LIN {X 0,Y 256.186,Z 305.925,A -85,B 0,C 180,E1 -18988.035,E2 -18988.035} C_VEL
LIN {X 0,Y 254.625,Z 317.423,A -85,B 0,C 180,E1 -18989.605,E2 -18989.605} C_VEL
LIN {X 0,Y 253.092,Z 328.163,A -85,B 0,C 180,E1 -18991.482,E2 -18991.482} C_VEL
LIN {X 0,Y 251.484,Z 337.845,A -85,B 0,C 180,E1 -18993.605,E2 -18993.605} C_VEL
LIN {X 0,Y 250.27,Z 345.355,A -85,B 0,C 180,E1 -18995.641,E2 -18995.641} C_VEL
LIN {X 0,Y 249.076,Z 352.738,A -85,B 0,C 180,E1 -18998.111,E2 -18998.111} C_VEL
LIN {X 0,Y 248.18,Z 358.597,A -85,B 0,C 180,E1 -19000.607,E2 -19000.607} C_VEL
LIN {X 0,Y 247.564,Z 363.197,A -85,B 0,C 180,E1 -19003.127,E2 -19003.127} C_VEL
LIN {X 0,Y 247.222,Z 365.688,A -85,B 0,C 180,E1 -19004.863,E2 -19004.863} C_VEL
LIN {X 0,Y 246.962,Z 367.629,A -85,B 0,C 180,E1 -19006.534,E2 -19006.534} C_VEL
LIN {X 0,Y 246.859,Z 369.106,A -85,B 0,C 180,E1 -19008.25,E2 -19008.25} C_VEL
LIN {X 0,Y 246.842,Z 370.181,A -85,B 0,C 180,E1 -19010.022,E2 -19010.022} C_VEL
LIN {X 0,Y 246.907,Z 370.793,A -85,B 0,C 180,E1 -19011.718,E2 -19011.718} C_VEL
LIN {X 0,Y 247.304,Z 370.822,A -85,B 0,C 180,E1 -19014.579,E2 -19014.579} C_VEL
LIN {X 0,Y 247.898,Z 369.931,A -85,B 0,C 180,E1 -19016.976,E2 -19016.976} C_VEL
LIN {X 0,Y 248.543,Z 368.668,A -85,B 0,C 180,E1 -19018.768,E2 -19018.768} C_VEL
LIN {X 0,Y 249.722,Z 365.952,A -85,B 0,C 180,E1 -19021.376,E2 -19021.376} C_VEL
LIN {X 0,Y 251.297,Z 362.009,A -85,B 0,C 180,E1 -19024.01,E2 -19024.01} C_VEL
LIN {X 0,Y 253.501,Z 356.251,A -85,B 0,C 180,E1 -19026.834,E2 -19026.834} C_VEL
LIN {X 0,Y 255.77,Z 349.911,A -85,B 0,C 180,E1 -19029.197,E2 -19029.197} C_VEL
LIN {X 0,Y 258.193,Z 342.787,A -85,B 0,C 180,E1 -19031.307,E2 -19031.307} C_VEL
LIN {X 0,Y 260.783,Z 334.381,A -85,B 0,C 180,E1 -19033.312,E2 -19033.312} C_VEL
LIN {X 0,Y 263.669,Z 324.355,A -85,B 0,C 180,E1 -19035.209,E2 -19035.209} C_VEL
LIN {X 0,Y 266.207,Z 314.054,A -85,B 0,C 180,E1 -19036.755,E2 -19036.755} C_VEL
LIN {X 0,Y 268.658,Z 301.667,A -85,B 0,C 180,E1 -19038.207,E2 -19038.207} C_VEL
LIN {X 0,Y 270.547,Z 289.737,A -85,B 0,C 180,E1 -19039.262,E2 -19039.262} C_VEL
LIN {X 0,Y 271.947,Z 277.419,A -85,B 0,C 180,E1 -19040.048,E2 -19040.048} C_VEL
LIN {X 0,Y 272.934,Z 264.372,A -85,B 0,C 180,E1 -19040.579,E2 -19040.579} C_VEL
LIN {X 0,Y 275.434,Z 209.115,A -85,B 0,C 180,E1 -19042.044,E2 -19042.044} C_VEL
LIN {X 0,Y 269.087,Z 195.685,A -85,B 0,C 180,E1 -19043.603,E2 -19043.603} C_VEL
LIN {X 0,Y 261.78,Z 182.263,A -85,B 0,C 180,E1 -19045.465,E2 -19045.465} C_VEL
LIN {X 0,Y 256.867,Z 174.801,A -85,B 0,C 180,E1 -19046.772,E2 -19046.772} C_VEL
LIN {X 0,Y 254.381,Z 171.129,A -85,B 0,C 180,E1 -19047.461,E2 -19047.461} C_VEL
LIN {X 0,Y 252.336,Z 167.962,A -85,B 0,C 180,E1 -19048.05,E2 -19048.05} C_VEL
LIN {X 0,Y 249.83,Z 164.955,A -85,B 0,C 180,E1 -19048.757,E2 -19048.757} C_VEL
LIN {X 0,Y 249.001,Z 162.468,A -85,B 0,C 180,E1 -19049.084,E2 -19049.084} C_VEL
LIN {X 0,Y 249.01,Z 162.471,A -85,B 0,C 180,E1 -19053.155,E2 -19053.155} C_VEL
LIN {X 0,Y 249.006,Z 162.464,A -85,B 0,C 180,E1 -19056.726,E2 -19056.726} C_VEL
LIN {X 0,Y 249.04,Z 162.458,A -85,B 0,C 180,E1 -19060.206,E2 -19060.206} C_VEL
LIN {X 0,Y 249.159,Z 162.446,A -85,B 0,C 180,E1 -19063.617,E2 -19063.617} C_VEL
LIN {X 0,Y 249.216,Z 162.429,A -85,B 0,C 180,E1 -19068.615,E2 -19068.615} C_VEL
LIN {X 0,Y 249.432,Z 162.411,A -85,B 0,C 180,E1 -19071.902,E2 -19071.902} C_VEL
LIN {X 0,Y 249.256,Z 162.433,A -85,B 0,C 180,E1 -19075.148,E2 -19075.148} C_VEL
LIN {X 0,Y 249.656,Z 162.371,A -85,B 0,C 180,E1 -19078.387,E2 -19078.387} C_VEL
LIN {X 0,Y 249.607,Z 162.381,A -85,B 0,C 180,E1 -19081.848,E2 -19081.848} C_VEL
LIN {X 0,Y 248.745,Z 162.486,A -85,B 0,C 180,E1 -19083.192,E2 -19083.192} C_VEL
LIN {X 0,Y 245.815,Z 162.865,A -85,B 0,C 180,E1 -19085.385,E2 -19085.385} C_VEL
LIN {X 0,Y 243.44,Z 163.151,A -85,B 0,C 180,E1 -19087.171,E2 -19087.171} C_VEL
LIN {X 0,Y 242.429,Z 163.273,A -85,B 0,C 180,E1 -19088.556,E2 -19088.556} C_VEL
LIN {X 0,Y 242.343,Z 163.287,A -85,B 0,C 180,E1 -19089.025,E2 -19089.025} C_VEL
LIN {X 0,Y 242.141,Z 163.308,A -85,B 0,C 180,E1 -19093.427,E2 -19093.427} C_VEL
LIN {X 0,Y 242.115,Z 163.314,A -85,B 0,C 180,E1 -19096.875,E2 -19096.875} C_VEL
LIN {X 0,Y 242.025,Z 163.323,A -85,B 0,C 180,E1 -19101.685,E2 -19101.685} C_VEL
LIN {X 0,Y 242.035,Z 163.326,A -85,B 0,C 180,E1 -19105.821,E2 -19105.821} C_VEL
LIN {X 0,Y 241.971,Z 163.337,A -85,B 0,C 180,E1 -19109.589,E2 -19109.589} C_VEL
LIN {X 0,Y 241.981,Z 163.336,A -85,B 0,C 180,E1 -19113.493,E2 -19113.493} C_VEL
LIN {X 0,Y 241.988,Z 163.335,A -85,B 0,C 180,E1 -19117.583,E2 -19117.583} C_VEL
LIN {X 0,Y 241.961,Z 163.345,A -85,B 0,C 180,E1 -19122.647,E2 -19122.647} C_VEL
LIN {X 0,Y 244.414,Z 171.283,A -85,B 0,C 180,E1 -19127.158,E2 -19127.158} C_VEL
LIN {X 0,Y 246.242,Z 177.579,A -85,B 0,C 180,E1 -19130.331,E2 -19130.331} C_VEL
LIN {X 0,Y 248.84,Z 182.168,A -85,B 0,C 180,E1 -19131.144,E2 -19131.144} C_VEL
LIN {X 0,Y 253.512,Z 190.412,A -85,B 0,C 180,E1 -19132.536,E2 -19132.536} C_VEL
LIN {X 0,Y 258.743,Z 200.398,A -85,B 0,C 180,E1 -19134.028,E2 -19134.028} C_VEL
LIN {X 0,Y 264.8,Z 213.402,A -85,B 0,C 180,E1 -19135.665,E2 -19135.665} C_VEL
LIN {X 0,Y 265.565,Z 216.293,A -85,B 0,C 180,E1 -19135.909,E2 -19135.909} C_VEL
LIN {X 0,Y 268.374,Z 234.977,A -85,B 0,C 180,E1 -19137.065,E2 -19137.065} C_VEL
LIN {X 0,Y 268.597,Z 238.665,A -85,B 0,C 180,E1 -19137.232,E2 -19137.232} C_VEL
LIN {X 0,Y 266.284,Z 287.985,A -85,B 0,C 180,E1 -19138.596,E2 -19138.596} C_VEL
LIN {X 0,Y 264.934,Z 300.799,A -85,B 0,C 180,E1 -19139.187,E2 -19139.187} C_VEL
LIN {X 0,Y 262.903,Z 313.363,A -85,B 0,C 180,E1 -19140.029,E2 -19140.029} C_VEL
LIN {X 0,Y 260.431,Z 325.458,A -85,B 0,C 180,E1 -19141.159,E2 -19141.159} C_VEL
LIN {X 0,Y 257.551,Z 336.958,A -85,B 0,C 180,E1 -19142.581,E2 -19142.581} C_VEL
LIN {X 0,Y 254.735,Z 347.328,A -85,B 0,C 180,E1 -19144.244,E2 -19144.244} C_VEL
LIN {X 0,Y 251.764,Z 356.728,A -85,B 0,C 180,E1 -19146.123,E2 -19146.123} C_VEL
LIN {X 0,Y 248.611,Z 365.821,A -85,B 0,C 180,E1 -19148.438,E2 -19148.438} C_VEL
LIN {X 0,Y 246.13,Z 373.27,A -85,B 0,C 180,E1 -19150.862,E2 -19150.862} C_VEL
LIN {X 0,Y 244.083,Z 379.142,A -85,B 0,C 180,E1 -19153.265,E2 -19153.265} C_VEL
LIN {X 0,Y 242.272,Z 383.877,A -85,B 0,C 180,E1 -19155.725,E2 -19155.725} C_VEL
LIN {X 0,Y 241.111,Z 387.528,A -85,B 0,C 180,E1 -19158.226,E2 -19158.226} C_VEL
LIN {X 0,Y 240.537,Z 389.435,A -85,B 0,C 180,E1 -19159.903,E2 -19159.903} C_VEL
LIN {X 0,Y 239.901,Z 391.944,A -85,B 0,C 180,E1 -19163.27,E2 -19163.27} C_VEL
LIN {X 0,Y 239.844,Z 392.655,A -85,B 0,C 180,E1 -19165.06,E2 -19165.06} C_VEL
LIN {X 0,Y 239.88,Z 392.916,A -85,B 0,C 180,E1 -19166.64,E2 -19166.64} C_VEL
LIN {X 0,Y 239.975,Z 392.787,A -85,B 0,C 180,E1 -19168.321,E2 -19168.321} C_VEL
LIN {X 0,Y 240.024,Z 392.244,A -85,B 0,C 180,E1 -19170,E2 -19170} C_VEL
LIN {X 0,Y 240,Z 391.3,A -85,B 0,C 180,E1 -19171.678,E2 -19171.678} C_VEL
LIN {X 0,Y 239.946,Z 389.947,A -85,B 0,C 180,E1 -19173.358,E2 -19173.358} C_VEL
LIN {X 0,Y 239.928,Z 387.153,A -85,B 0,C 180,E1 -19175.8,E2 -19175.8} C_VEL
LIN {X 0,Y 240.145,Z 383.08,A -85,B 0,C 180,E1 -19178.414,E2 -19178.414} C_VEL
LIN {X 0,Y 240.752,Z 376.941,A -85,B 0,C 180,E1 -19181.364,E2 -19181.364} C_VEL
LIN {X 0,Y 241.739,Z 370.201,A -85,B 0,C 180,E1 -19183.877,E2 -19183.877} C_VEL
LIN {X 0,Y 243.075,Z 361.811,A -85,B 0,C 180,E1 -19186.373,E2 -19186.373} C_VEL
LIN {X 0,Y 244.362,Z 353.148,A -85,B 0,C 180,E1 -19188.443,E2 -19188.443} C_VEL
LIN {X 0,Y 245.985,Z 343.66,A -85,B 0,C 180,E1 -19190.268,E2 -19190.268} C_VEL
LIN {X 0,Y 247.537,Z 333.302,A -85,B 0,C 180,E1 -19191.878,E2 -19191.878} C_VEL
LIN {X 0,Y 249.154,Z 321.996,A -85,B 0,C 180,E1 -19193.26,E2 -19193.26} C_VEL
LIN {X 0,Y 250.656,Z 309.271,A -85,B 0,C 180,E1 -19194.429,E2 -19194.429} C_VEL
LIN {X 0,Y 251.789,Z 296.575,A -85,B 0,C 180,E1 -19195.248,E2 -19195.248} C_VEL
LIN {X 0,Y 252.504,Z 283.619,A -85,B 0,C 180,E1 -19195.778,E2 -19195.778} C_VEL
LIN {X 0,Y 253.878,Z 231.504,A -85,B 0,C 180,E1 -19197.262,E2 -19197.262} C_VEL
LIN {X 0,Y 248.722,Z 189.37,A -85,B 0,C 180,E1 -19199.055,E2 -19199.055} C_VEL
LIN {X 0,Y 245.558,Z 179.931,A -85,B 0,C 180,E1 -19199.718,E2 -19199.718} C_VEL
LIN {X 0,Y 243.224,Z 168.679,A -85,B 0,C 180,E1 -19203.795,E2 -19203.795} C_VEL
LIN {X 0,Y 242.065,Z 163.335,A -85,B 0,C 180,E1 -19205.868,E2 -19205.868} C_VEL
LIN {X 0,Y 241.973,Z 163.346,A -85,B 0,C 180,E1 -19209.715,E2 -19209.715} C_VEL
LIN {X 0,Y 241.931,Z 163.35,A -85,B 0,C 180,E1 -19214.202,E2 -19214.202} C_VEL
LIN {X 0,Y 241.938,Z 163.35,A -85,B 0,C 180,E1 -19218.077,E2 -19218.077} C_VEL
LIN {X 0,Y 241.991,Z 163.341,A -85,B 0,C 180,E1 -19222.418,E2 -19222.418} C_VEL
LIN {X 0,Y 241.988,Z 163.341,A -85,B 0,C 180,E1 -19226.508,E2 -19226.508} C_VEL
LIN {X 0,Y 242.038,Z 163.335,A -85,B 0,C 180,E1 -19230.587,E2 -19230.587} C_VEL
LIN {X 0,Y 242.068,Z 163.33,A -85,B 0,C 180,E1 -19234.183,E2 -19234.183} C_VEL
LIN {X 0,Y 242.024,Z 163.331,A -85,B 0,C 180,E1 -19238.315,E2 -19238.315} C_VEL
LIN {X 0,Y 242.115,Z 163.303,A -85,B 0,C 180,E1 -19243.316,E2 -19243.316} C_VEL
LIN {X 0,Y 242.167,Z 163.316,A -85,B 0,C 180,E1 -19248.278,E2 -19248.278} C_VEL
LIN {X 0,Y 242.372,Z 163.288,A -85,B 0,C 180,E1 -19251.663,E2 -19251.663} C_VEL
LIN {X 0,Y 242.246,Z 163.304,A -85,B 0,C 180,E1 -19255.007,E2 -19255.007} C_VEL
LIN {X 0,Y 242.635,Z 163.259,A -85,B 0,C 180,E1 -19258.34,E2 -19258.34} C_VEL
LIN {X 0,Y 242.636,Z 163.25,A -85,B 0,C 180,E1 -19261.659,E2 -19261.659} C_VEL
LIN {X 0,Y 242.421,Z 163.287,A -85,B 0,C 180,E1 -19266.683,E2 -19266.683} C_VEL
LIN {X 0,Y 242.267,Z 163.302,A -85,B 0,C 180,E1 -19270.023,E2 -19270.023} C_VEL
LIN {X 0,Y 242.166,Z 163.317,A -85,B 0,C 180,E1 -19275.14,E2 -19275.14} C_VEL
LIN {X 0,Y 242.071,Z 163.327,A -85,B 0,C 180,E1 -19278.624,E2 -19278.624} C_VEL
LIN {X 0,Y 242.006,Z 163.332,A -85,B 0,C 180,E1 -19282.18,E2 -19282.18} C_VEL
LIN {X 0,Y 242.066,Z 163.332,A -85,B 0,C 180,E1 -19285.838,E2 -19285.838} C_VEL
LIN {X 0,Y 242.006,Z 163.333,A -85,B 0,C 180,E1 -19289.583,E2 -19289.583} C_VEL
LIN {X 0,Y 241.98,Z 163.339,A -85,B 0,C 180,E1 -19293.492,E2 -19293.492} C_VEL
LIN {X 0,Y 241.991,Z 163.335,A -85,B 0,C 180,E1 -19297.581,E2 -19297.581} C_VEL
LIN {X 0,Y 241.936,Z 163.348,A -85,B 0,C 180,E1 -19301.922,E2 -19301.922} C_VEL
LIN {X 0,Y 241.933,Z 163.344,A -85,B 0,C 180,E1 -19306.571,E2 -19306.571} C_VEL
LIN {X 0,Y 241.955,Z 163.342,A -85,B 0,C 180,E1 -19310.281,E2 -19310.281} C_VEL
LIN {X 0,Y 241.987,Z 163.34,A -85,B 0,C 180,E1 -19314.489,E2 -19314.489} C_VEL
LIN {X 0,Y 241.973,Z 163.33,A -85,B 0,C 180,E1 -19318.48,E2 -19318.48} C_VEL
LIN {X 0,Y 242.007,Z 163.339,A -85,B 0,C 180,E1 -19322.313,E2 -19322.313} C_VEL
LIN {X 0,Y 242.04,Z 163.328,A -85,B 0,C 180,E1 -19326.014,E2 -19326.014} C_VEL
LIN {X 0,Y 242.021,Z 163.337,A -85,B 0,C 180,E1 -19329.607,E2 -19329.607} C_VEL
LIN {X 0,Y 242.127,Z 163.326,A -85,B 0,C 180,E1 -19333.307,E2 -19333.307} C_VEL
LIN {X 0,Y 242.167,Z 163.318,A -85,B 0,C 180,E1 -19338.279,E2 -19338.279} C_VEL
LIN {X 0,Y 242.31,Z 163.301,A -85,B 0,C 180,E1 -19340.186,E2 -19340.186} C_VEL
LIN {X 0,Y 243.419,Z 166.268,A -85,B 0,C 180,E1 -19340.407,E2 -19340.407} C_VEL
LIN {X 0,Y 249.348,Z 179.959,A -85,B 0,C 180,E1 -19341.447,E2 -19341.447} C_VEL
LIN {X 0,Y 254.912,Z 195.622,A -85,B 0,C 180,E1 -19342.468,E2 -19342.468} C_VEL
LIN {X 0,Y 252.621,Z 267.383,A -85,B 0,C 180,E1 -19344.513,E2 -19344.513} C_VEL
LIN {X 0,Y 251.839,Z 280.568,A -85,B 0,C 180,E1 -19345.198,E2 -19345.198} C_VEL
LIN {X 0,Y 250.849,Z 293.258,A -85,B 0,C 180,E1 -19346.185,E2 -19346.185} C_VEL
LIN {X 0,Y 249.624,Z 304.622,A -85,B 0,C 180,E1 -19347.378,E2 -19347.378} C_VEL
LIN {X 0,Y 248.002,Z 316.41,A -85,B 0,C 180,E1 -19348.985,E2 -19348.985} C_VEL
LIN {X 0,Y 246.436,Z 326.966,A -85,B 0,C 180,E1 -19350.813,E2 -19350.813} C_VEL
LIN {X 0,Y 244.821,Z 336.495,A -85,B 0,C 180,E1 -19352.88,E2 -19352.88} C_VEL
LIN {X 0,Y 243.458,Z 344.296,A -85,B 0,C 180,E1 -19354.968,E2 -19354.968} C_VEL
LIN {X 0,Y 242.229,Z 351.914,A -85,B 0,C 180,E1 -19357.502,E2 -19357.502} C_VEL
LIN {X 0,Y 241.248,Z 358.034,A -85,B 0,C 180,E1 -19360.067,E2 -19360.067} C_VEL
LIN {X 0,Y 240.564,Z 362.854,A -85,B 0,C 180,E1 -19362.657,E2 -19362.657} C_VEL
LIN {X 0,Y 240.065,Z 366.523,A -85,B 0,C 180,E1 -19365.277,E2 -19365.277} C_VEL
LIN {X 0,Y 239.812,Z 368.353,A -85,B 0,C 180,E1 -19367.042,E2 -19367.042} C_VEL
LIN {X 0,Y 239.757,Z 370.554,A -85,B 0,C 180,E1 -19370.28,E2 -19370.28} C_VEL
LIN {X 0,Y 239.889,Z 371.185,A -85,B 0,C 180,E1 -19372.387,E2 -19372.387} C_VEL
LIN {X 0,Y 240.292,Z 371.134,A -85,B 0,C 180,E1 -19374.95,E2 -19374.95} C_VEL
LIN {X 0,Y 241.065,Z 369.98,A -85,B 0,C 180,E1 -19377.805,E2 -19377.805} C_VEL
LIN {X 0,Y 241.77,Z 368.645,A -85,B 0,C 180,E1 -19379.615,E2 -19379.615} C_VEL
LIN {X 0,Y 243.144,Z 365.714,A -85,B 0,C 180,E1 -19382.326,E2 -19382.326} C_VEL
LIN {X 0,Y 244.869,Z 361.57,A -85,B 0,C 180,E1 -19385.031,E2 -19385.031} C_VEL
LIN {X 0,Y 247.129,Z 355.995,A -85,B 0,C 180,E1 -19387.715,E2 -19387.715} C_VEL
LIN {X 0,Y 249.796,Z 348.922,A -85,B 0,C 180,E1 -19390.324,E2 -19390.324} C_VEL
LIN {X 0,Y 252.388,Z 341.533,A -85,B 0,C 180,E1 -19392.475,E2 -19392.475} C_VEL
LIN {X 0,Y 255.07,Z 333.222,A -85,B 0,C 180,E1 -19394.423,E2 -19394.423} C_VEL
LIN {X 0,Y 257.925,Z 323.554,A -85,B 0,C 180,E1 -19396.227,E2 -19396.227} C_VEL
LIN {X 0,Y 260.811,Z 312.036,A -85,B 0,C 180,E1 -19397.912,E2 -19397.912} C_VEL
LIN {X 0,Y 263.129,Z 300.167,A -85,B 0,C 180,E1 -19399.278,E2 -19399.278} C_VEL
LIN {X 0,Y 265.155,Z 287.446,A -85,B 0,C 180,E1 -19400.34,E2 -19400.34} C_VEL
LIN {X 0,Y 266.636,Z 274.106,A -85,B 0,C 180,E1 -19401.127,E2 -19401.127} C_VEL
LIN {X 0,Y 267.546,Z 260.182,A -85,B 0,C 180,E1 -19401.614,E2 -19401.614} C_VEL
LIN {X 0,Y 269.806,Z 211.318,A -85,B 0,C 180,E1 -19402.926,E2 -19402.926} C_VEL
LIN {X 0,Y 263.658,Z 198.379,A -85,B 0,C 180,E1 -19404.506,E2 -19404.506} C_VEL
LIN {X 0,Y 256.375,Z 184.98,A -85,B 0,C 180,E1 -19406.478,E2 -19406.478} C_VEL
LIN {X 0,Y 250.23,Z 176.008,A -85,B 0,C 180,E1 -19408.203,E2 -19408.203} C_VEL
LIN {X 0,Y 247.673,Z 172.35,A -85,B 0,C 180,E1 -19408.96,E2 -19408.96} C_VEL
LIN {X 0,Y 245.475,Z 169.112,A -85,B 0,C 180,E1 -19409.636,E2 -19409.636} C_VEL
LIN {X 0,Y 244.526,Z 167.97,A -85,B 0,C 180,E1 -19409.923,E2 -19409.923} C_VEL
LIN {X 0,Y 242.653,Z 165.642,A -85,B 0,C 180,E1 -19410.504,E2 -19410.504} C_VEL
LIN {X 0,Y 241.976,Z 163.343,A -85,B 0,C 180,E1 -19410.815,E2 -19410.815} C_VEL
LIN {X 0,Y 241.996,Z 163.337,A -85,B 0,C 180,E1 -19414.198,E2 -19414.198} C_VEL
LIN {X 0,Y 241.986,Z 163.337,A -85,B 0,C 180,E1 -19418.339,E2 -19418.339} C_VEL
LIN {X 0,Y 242.107,Z 163.328,A -85,B 0,C 180,E1 -19423.325,E2 -19423.325} C_VEL
LIN {X 0,Y 242.15,Z 163.311,A -85,B 0,C 180,E1 -19428.278,E2 -19428.278} C_VEL
LIN {X 0,Y 242.382,Z 163.292,A -85,B 0,C 180,E1 -19431.664,E2 -19431.664} C_VEL
LIN {X 0,Y 242.401,Z 163.276,A -85,B 0,C 180,E1 -19433.341,E2 -19433.341} C_VEL
LIN {X 0,Y 242.616,Z 163.247,A -85,B 0,C 180,E1 -19438.34,E2 -19438.34} C_VEL
LIN {X 0,Y 242.595,Z 163.255,A -85,B 0,C 180,E1 -19441.76,E2 -19441.76} C_VEL
LIN {X 0,Y 242.398,Z 163.282,A -85,B 0,C 180,E1 -19446.66,E2 -19446.66} C_VEL
LIN {X 0,Y 242.343,Z 163.287,A -85,B 0,C 180,E1 -19449.025,E2 -19449.025} C_VEL
LIN {X 0,Y 241.643,Z 163.386,A -85,B 0,C 180,E1 -19450.411,E2 -19450.411} C_VEL
LIN {X 0,Y 238.702,Z 163.758,A -85,B 0,C 180,E1 -19452.668,E2 -19452.668} C_VEL
LIN {X 0,Y 236.212,Z 164.064,A -85,B 0,C 180,E1 -19454.508,E2 -19454.508} C_VEL
LIN {X 0,Y 235.146,Z 164.192,A -85,B 0,C 180,E1 -19455.938,E2 -19455.938} C_VEL
LIN {X 0,Y 235.06,Z 164.195,A -85,B 0,C 180,E1 -19456.424,E2 -19456.424} C_VEL
LIN {X 0,Y 234.994,Z 164.204,A -85,B 0,C 180,E1 -19461.032,E2 -19461.032} C_VEL
LIN {X 0,Y 234.971,Z 164.203,A -85,B 0,C 180,E1 -19466.194,E2 -19466.194} C_VEL
LIN {X 0,Y 234.901,Z 164.214,A -85,B 0,C 180,E1 -19470.573,E2 -19470.573} C_VEL
LIN {X 0,Y 234.932,Z 164.213,A -85,B 0,C 180,E1 -19474.638,E2 -19474.638} C_VEL
LIN {X 0,Y 234.914,Z 164.225,A -85,B 0,C 180,E1 -19478.935,E2 -19478.935} C_VEL
LIN {X 0,Y 234.894,Z 164.364,A -85,B 0,C 180,E1 -19481.024,E2 -19481.024} C_VEL
LIN {X 0,Y 237.142,Z 171.449,A -85,B 0,C 180,E1 -19485.339,E2 -19485.339} C_VEL
LIN {X 0,Y 238.91,Z 177.249,A -85,B 0,C 180,E1 -19488.443,E2 -19488.443} C_VEL
LIN {X 0,Y 241.514,Z 181.66,A -85,B 0,C 180,E1 -19489.329,E2 -19489.329} C_VEL
LIN {X 0,Y 246.23,Z 189.555,A -85,B 0,C 180,E1 -19490.838,E2 -19490.838} C_VEL
LIN {X 0,Y 251.063,Z 198.309,A -85,B 0,C 180,E1 -19492.314,E2 -19492.314} C_VEL
LIN {X 0,Y 257.044,Z 210.58,A -85,B 0,C 180,E1 -19494.072,E2 -19494.072} C_VEL
LIN {X 0,Y 260.198,Z 218.145,A -85,B 0,C 180,E1 -19494.976,E2 -19494.976} C_VEL
LIN {X 0,Y 262.902,Z 236.53,A -85,B 0,C 180,E1 -19496.153,E2 -19496.153} C_VEL
LIN {X 0,Y 263.057,Z 239.658,A -85,B 0,C 180,E1 -19496.293,E2 -19496.293} C_VEL
LIN {X 0,Y 260.67,Z 287.976,A -85,B 0,C 180,E1 -19497.655,E2 -19497.655} C_VEL
LIN {X 0,Y 259.243,Z 300.794,A -85,B 0,C 180,E1 -19498.258,E2 -19498.258} C_VEL
LIN {X 0,Y 257.04,Z 313.88,A -85,B 0,C 180,E1 -19499.158,E2 -19499.158} C_VEL
LIN {X 0,Y 254.675,Z 324.942,A -85,B 0,C 180,E1 -19500.216,E2 -19500.216} C_VEL
LIN {X 0,Y 251.673,Z 336.477,A -85,B 0,C 180,E1 -19501.658,E2 -19501.658} C_VEL
LIN {X 0,Y 248.716,Z 346.875,A -85,B 0,C 180,E1 -19503.347,E2 -19503.347} C_VEL
LIN {X 0,Y 245.882,Z 355.42,A -85,B 0,C 180,E1 -19505.064,E2 -19505.064} C_VEL
LIN {X 0,Y 243.045,Z 363.328,A -85,B 0,C 180,E1 -19507.022,E2 -19507.022} C_VEL
LIN {X 0,Y 240.228,Z 371.107,A -85,B 0,C 180,E1 -19509.447,E2 -19509.447} C_VEL
LIN {X 0,Y 237.96,Z 377.373,A -85,B 0,C 180,E1 -19511.934,E2 -19511.934} C_VEL
LIN {X 0,Y 235.959,Z 382.398,A -85,B 0,C 180,E1 -19514.451,E2 -19514.451} C_VEL
LIN {X 0,Y 234.446,Z 386.325,A -85,B 0,C 180,E1 -19517.007,E2 -19517.007} C_VEL
LIN {X 0,Y 233.522,Z 389.261,A -85,B 0,C 180,E1 -19519.596,E2 -19519.596} C_VEL
LIN {X 0,Y 232.822,Z 391.697,A -85,B 0,C 180,E1 -19523.065,E2 -19523.065} C_VEL
LIN {X 0,Y 232.773,Z 392.426,A -85,B 0,C 180,E1 -19525.111,E2 -19525.111} C_VEL
LIN {X 0,Y 232.902,Z 392.413,A -85,B 0,C 180,E1 -19528.27,E2 -19528.27} C_VEL
LIN {X 0,Y 232.951,Z 391.839,A -85,B 0,C 180,E1 -19530,E2 -19530} C_VEL
LIN {X 0,Y 232.928,Z 390.863,A -85,B 0,C 180,E1 -19531.729,E2 -19531.729} C_VEL
LIN {X 0,Y 232.864,Z 389.463,A -85,B 0,C 180,E1 -19533.46,E2 -19533.46} C_VEL
LIN {X 0,Y 232.841,Z 386.498,A -85,B 0,C 180,E1 -19536.064,E2 -19536.064} C_VEL
LIN {X 0,Y 233.092,Z 382.46,A -85,B 0,C 180,E1 -19538.67,E2 -19538.67} C_VEL
LIN {X 0,Y 233.746,Z 376.203,A -85,B 0,C 180,E1 -19541.709,E2 -19541.709} C_VEL
LIN {X 0,Y 234.812,Z 369.373,A -85,B 0,C 180,E1 -19544.295,E2 -19544.295} C_VEL
LIN {X 0,Y 236.238,Z 360.854,A -85,B 0,C 180,E1 -19546.861,E2 -19546.861} C_VEL
LIN {X 0,Y 237.384,Z 353.158,A -85,B 0,C 180,E1 -19548.747,E2 -19548.747} C_VEL
LIN {X 0,Y 239.085,Z 343.561,A -85,B 0,C 180,E1 -19550.655,E2 -19550.655} C_VEL
LIN {X 0,Y 240.688,Z 333.251,A -85,B 0,C 180,E1 -19552.308,E2 -19552.308} C_VEL
LIN {X 0,Y 242.359,Z 322.011,A -85,B 0,C 180,E1 -19553.725,E2 -19553.725} C_VEL
LIN {X 0,Y 243.904,Z 309.441,A -85,B 0,C 180,E1 -19554.923,E2 -19554.923} C_VEL
LIN {X 0,Y 245.142,Z 296.032,A -85,B 0,C 180,E1 -19555.811,E2 -19555.811} C_VEL
LIN {X 0,Y 245.885,Z 282.94,A -85,B 0,C 180,E1 -19556.354,E2 -19556.354} C_VEL
LIN {X 0,Y 247.259,Z 232.291,A -85,B 0,C 180,E1 -19557.833,E2 -19557.833} C_VEL
LIN {X 0,Y 242.359,Z 191.437,A -85,B 0,C 180,E1 -19559.625,E2 -19559.625} C_VEL
LIN {X 0,Y 238.245,Z 179.646,A -85,B 0,C 180,E1 -19560.472,E2 -19560.472} C_VEL
LIN {X 0,Y 236.063,Z 169.033,A -85,B 0,C 180,E1 -19564.448,E2 -19564.448} C_VEL
LIN {X 0,Y 235.005,Z 164.217,A -85,B 0,C 180,E1 -19566.372,E2 -19566.372} C_VEL
LIN {X 0,Y 234.943,Z 164.22,A -85,B 0,C 180,E1 -19568.944,E2 -19568.944} C_VEL
LIN {X 0,Y 234.888,Z 164.228,A -85,B 0,C 180,E1 -19573.485,E2 -19573.485} C_VEL
LIN {X 0,Y 234.888,Z 164.226,A -85,B 0,C 180,E1 -19576.514,E2 -19576.514} C_VEL
LIN {X 0,Y 234.919,Z 164.224,A -85,B 0,C 180,E1 -19581.078,E2 -19581.078} C_VEL
LIN {X 0,Y 234.943,Z 164.222,A -85,B 0,C 180,E1 -19585.364,E2 -19585.364} C_VEL
LIN {X 0,Y 234.933,Z 164.222,A -85,B 0,C 180,E1 -19589.432,E2 -19589.432} C_VEL
LIN {X 0,Y 234.995,Z 164.212,A -85,B 0,C 180,E1 -19593.793,E2 -19593.793} C_VEL
LIN {X 0,Y 234.99,Z 164.203,A -85,B 0,C 180,E1 -19598.967,E2 -19598.967} C_VEL
LIN {X 0,Y 235.056,Z 164.178,A -85,B 0,C 180,E1 -19603.092,E2 -19603.092} C_VEL
LIN {X 0,Y 235.099,Z 164.196,A -85,B 0,C 180,E1 -19607.921,E2 -19607.921} C_VEL
LIN {X 0,Y 235.312,Z 164.168,A -85,B 0,C 180,E1 -19611.411,E2 -19611.411} C_VEL
LIN {X 0,Y 235.206,Z 164.179,A -85,B 0,C 180,E1 -19614.857,E2 -19614.857} C_VEL
LIN {X 0,Y 235.594,Z 164.135,A -85,B 0,C 180,E1 -19618.29,E2 -19618.29} C_VEL
LIN {X 0,Y 235.595,Z 164.127,A -85,B 0,C 180,E1 -19621.709,E2 -19621.709} C_VEL
LIN {X 0,Y 235.373,Z 164.164,A -85,B 0,C 180,E1 -19626.859,E2 -19626.859} C_VEL
LIN {X 0,Y 235.214,Z 164.177,A -85,B 0,C 180,E1 -19630.327,E2 -19630.327} C_VEL
LIN {X 0,Y 235.113,Z 164.196,A -85,B 0,C 180,E1 -19635.606,E2 -19635.606} C_VEL
LIN {X 0,Y 235.007,Z 164.205,A -85,B 0,C 180,E1 -19639.205,E2 -19639.205} C_VEL
LIN {X 0,Y 234.952,Z 164.213,A -85,B 0,C 180,E1 -19642.883,E2 -19642.883} C_VEL
LIN {X 0,Y 234.966,Z 164.214,A -85,B 0,C 180,E1 -19646.657,E2 -19646.657} C_VEL
LIN {X 0,Y 234.921,Z 164.213,A -85,B 0,C 180,E1 -19650.569,E2 -19650.569} C_VEL
LIN {X 0,Y 234.932,Z 164.217,A -85,B 0,C 180,E1 -19654.637,E2 -19654.637} C_VEL
LIN {X 0,Y 234.941,Z 164.21,A -85,B 0,C 180,E1 -19658.944,E2 -19658.944} C_VEL
LIN {X 0,Y 234.886,Z 164.225,A -85,B 0,C 180,E1 -19663.486,E2 -19663.486} C_VEL
LIN {X 0,Y 234.886,Z 164.221,A -85,B 0,C 180,E1 -19666.514,E2 -19666.514} C_VEL
LIN {X 0,Y 234.917,Z 164.219,A -85,B 0,C 180,E1 -19671.079,E2 -19671.079} C_VEL
LIN {X 0,Y 234.929,Z 164.221,A -85,B 0,C 180,E1 -19675.362,E2 -19675.362} C_VEL
LIN {X 0,Y 234.931,Z 164.21,A -85,B 0,C 180,E1 -19679.433,E2 -19679.433} C_VEL
LIN {X 0,Y 234.993,Z 164.211,A -85,B 0,C 180,E1 -19683.794,E2 -19683.794} C_VEL
LIN {X 0,Y 234.99,Z 164.216,A -85,B 0,C 180,E1 -19688.968,E2 -19688.968} C_VEL
LIN {X 0,Y 235.063,Z 164.206,A -85,B 0,C 180,E1 -19693.086,E2 -19693.086} C_VEL
LIN {X 0,Y 235.099,Z 164.198,A -85,B 0,C 180,E1 -19697.922,E2 -19697.922} C_VEL
LIN {X 0,Y 235.19,Z 164.316,A -85,B 0,C 180,E1 -19699.456,E2 -19699.456} C_VEL
LIN {X 0,Y 236.375,Z 167.291,A -85,B 0,C 180,E1 -19699.689,E2 -19699.689} C_VEL
LIN {X 0,Y 242.76,Z 181.381,A -85,B 0,C 180,E1 -19700.833,E2 -19700.833} C_VEL
LIN {X 0,Y 248.446,Z 197.561,A -85,B 0,C 180,E1 -19701.919,E2 -19701.919} C_VEL
LIN {X 0,Y 245.973,Z 267.685,A -85,B 0,C 180,E1 -19703.952,E2 -19703.952} C_VEL
LIN {X 0,Y 245.168,Z 280.867,A -85,B 0,C 180,E1 -19704.655,E2 -19704.655} C_VEL
LIN {X 0,Y 244.12,Z 293.574,A -85,B 0,C 180,E1 -19705.666,E2 -19705.666} C_VEL
LIN {X 0,Y 242.852,Z 304.938,A -85,B 0,C 180,E1 -19706.89,E2 -19706.89} C_VEL
LIN {X 0,Y 241.183,Z 316.723,A -85,B 0,C 180,E1 -19708.539,E2 -19708.539} C_VEL
LIN {X 0,Y 239.489,Z 327.811,A -85,B 0,C 180,E1 -19710.522,E2 -19710.522} C_VEL
LIN {X 0,Y 237.875,Z 336.816,A -85,B 0,C 180,E1 -19712.54,E2 -19712.54} C_VEL
LIN {X 0,Y 236.491,Z 344.611,A -85,B 0,C 180,E1 -19714.688,E2 -19714.688} C_VEL
LIN {X 0,Y 235.189,Z 352.237,A -85,B 0,C 180,E1 -19717.297,E2 -19717.297} C_VEL
LIN {X 0,Y 234.201,Z 358.262,A -85,B 0,C 180,E1 -19719.893,E2 -19719.893} C_VEL
LIN {X 0,Y 233.564,Z 362.437,A -85,B 0,C 180,E1 -19722.16,E2 -19722.16} C_VEL
LIN {X 0,Y 232.98,Z 366.647,A -85,B 0,C 180,E1 -19725.139,E2 -19725.139} C_VEL
LIN {X 0,Y 232.702,Z 369.068,A -85,B 0,C 180,E1 -19727.579,E2 -19727.579} C_VEL
LIN {X 0,Y 232.665,Z 370.923,A -85,B 0,C 180,E1 -19730.545,E2 -19730.545} C_VEL
LIN {X 0,Y 232.865,Z 371.57,A -85,B 0,C 180,E1 -19733.101,E2 -19733.101} C_VEL
LIN {X 0,Y 233.272,Z 371.449,A -85,B 0,C 180,E1 -19735.334,E2 -19735.334} C_VEL
LIN {X 0,Y 234.285,Z 370.019,A -85,B 0,C 180,E1 -19738.683,E2 -19738.683} C_VEL
LIN {X 0,Y 235.089,Z 368.589,A -85,B 0,C 180,E1 -19740.545,E2 -19740.545} C_VEL
LIN {X 0,Y 236.938,Z 364.729,A -85,B 0,C 180,E1 -19743.847,E2 -19743.847} C_VEL
LIN {X 0,Y 239.219,Z 359.541,A -85,B 0,C 180,E1 -19746.92,E2 -19746.92} C_VEL
LIN {X 0,Y 241.915,Z 353.06,A -85,B 0,C 180,E1 -19749.728,E2 -19749.728} C_VEL
LIN {X 0,Y 245.026,Z 345.064,A -85,B 0,C 180,E1 -19752.38,E2 -19752.38} C_VEL
LIN {X 0,Y 247.914,Z 336.72,A -85,B 0,C 180,E1 -19754.558,E2 -19754.558} C_VEL
LIN {X 0,Y 250.872,Z 327.605,A -85,B 0,C 180,E1 -19756.429,E2 -19756.429} C_VEL
LIN {X 0,Y 253.706,Z 317.379,A -85,B 0,C 180,E1 -19758.114,E2 -19758.114} C_VEL
LIN {X 0,Y 256.214,Z 306.701,A -85,B 0,C 180,E1 -19759.509,E2 -19759.509} C_VEL
LIN {X 0,Y 258.346,Z 295.263,A -85,B 0,C 180,E1 -19760.68,E2 -19760.68} C_VEL
LIN {X 0,Y 260.16,Z 282.405,A -85,B 0,C 180,E1 -19761.636,E2 -19761.636} C_VEL
LIN {X 0,Y 261.503,Z 268.62,A -85,B 0,C 180,E1 -19762.316,E2 -19762.316} C_VEL
LIN {X 0,Y 264.324,Z 213.887,A -85,B 0,C 180,E1 -19763.818,E2 -19763.818} C_VEL
LIN {X 0,Y 258.714,Z 201.979,A -85,B 0,C 180,E1 -19765.335,E2 -19765.335} C_VEL
LIN {X 0,Y 252.625,Z 190.521,A -85,B 0,C 180,E1 -19767.07,E2 -19767.07} C_VEL
LIN {X 0,Y 246.332,Z 181.121,A -85,B 0,C 180,E1 -19768.91,E2 -19768.91} C_VEL
LIN {X 0,Y 243.698,Z 177.358,A -85,B 0,C 180,E1 -19769.72,E2 -19769.72} C_VEL
LIN {X 0,Y 240.949,Z 173.51,A -85,B 0,C 180,E1 -19770.596,E2 -19770.596} C_VEL
LIN {X 0,Y 238.776,Z 170.51,A -85,B 0,C 180,E1 -19771.324,E2 -19771.324} C_VEL
LIN {X 0,Y 238.195,Z 169.351,A -85,B 0,C 180,E1 -19771.54,E2 -19771.54} C_VEL
LIN {X 0,Y 235.987,Z 167.2,A -85,B 0,C 180,E1 -19772.269,E2 -19772.269} C_VEL
LIN {X 0,Y 234.977,Z 164.73,A -85,B 0,C 180,E1 -19772.683,E2 -19772.683} C_VEL
LIN {X 0,Y 234.917,Z 164.229,A -85,B 0,C 180,E1 -19772.796,E2 -19772.796} C_VEL
LIN {X 0,Y 234.916,Z 164.217,A -85,B 0,C 180,E1 -19777.113,E2 -19777.113} C_VEL
LIN {X 0,Y 234.957,Z 164.209,A -85,B 0,C 180,E1 -19780.79,E2 -19780.79} C_VEL
LIN {X 0,Y 235.04,Z 164.197,A -85,B 0,C 180,E1 -19784.389,E2 -19784.389} C_VEL
LIN {X 0,Y 235.184,Z 164.177,A -85,B 0,C 180,E1 -19789.671,E2 -19789.671} C_VEL
LIN {X 0,Y 235.353,Z 164.154,A -85,B 0,C 180,E1 -19793.14,E2 -19793.14} C_VEL
LIN {X 0,Y 235.575,Z 164.124,A -85,B 0,C 180,E1 -19798.291,E2 -19798.291} C_VEL
LIN {X 0,Y 235.577,Z 164.13,A -85,B 0,C 180,E1 -19801.71,E2 -19801.71} C_VEL
LIN {X 0,Y 235.35,Z 164.157,A -85,B 0,C 180,E1 -19806.861,E2 -19806.861} C_VEL
LIN {X 0,Y 235.214,Z 164.186,A -85,B 0,C 180,E1 -19810.328,E2 -19810.328} C_VEL
LIN {X 0,Y 235.088,Z 164.201,A -85,B 0,C 180,E1 -19815.609,E2 -19815.609} C_VEL
LIN {X 0,Y 235.06,Z 164.195,A -85,B 0,C 180,E1 -19816.424,E2 -19816.424} C_VEL
LIN {X 0,Y 234.389,Z 164.276,A -85,B 0,C 180,E1 -19817.853,E2 -19817.853} C_VEL
LIN {X 0,Y 231.511,Z 164.646,A -85,B 0,C 180,E1 -19820.183,E2 -19820.183} C_VEL
LIN {X 0,Y 229.049,Z 164.951,A -85,B 0,C 180,E1 -19822.083,E2 -19822.083} C_VEL
LIN {X 0,Y 227.974,Z 165.079,A -85,B 0,C 180,E1 -19823.559,E2 -19823.559} C_VEL
LIN {X 0,Y 227.876,Z 165.088,A -85,B 0,C 180,E1 -19824.06,E2 -19824.06} C_VEL
LIN {X 0,Y 227.858,Z 165.093,A -85,B 0,C 180,E1 -19827.559,E2 -19827.559} C_VEL
LIN {X 0,Y 227.858,Z 165.096,A -85,B 0,C 180,E1 -19831.625,E2 -19831.625} C_VEL
LIN {X 0,Y 227.883,Z 165.1,A -85,B 0,C 180,E1 -19835.872,E2 -19835.872} C_VEL
LIN {X 0,Y 227.882,Z 165.244,A -85,B 0,C 180,E1 -19839.121,E2 -19839.121} C_VEL
LIN {X 0,Y 229.958,Z 171.78,A -85,B 0,C 180,E1 -19843.443,E2 -19843.443} C_VEL
LIN {X 0,Y 231.512,Z 176.712,A -85,B 0,C 180,E1 -19846.286,E2 -19846.286} C_VEL
LIN {X 0,Y 234.646,Z 181.699,A -85,B 0,C 180,E1 -19847.458,E2 -19847.458} C_VEL
LIN {X 0,Y 239.621,Z 189.953,A -85,B 0,C 180,E1 -19849.21,E2 -19849.21} C_VEL
LIN {X 0,Y 242.753,Z 195.373,A -85,B 0,C 180,E1 -19850.243,E2 -19850.243} C_VEL
LIN {X 0,Y 248.719,Z 206.665,A -85,B 0,C 180,E1 -19852.129,E2 -19852.129} C_VEL
LIN {X 0,Y 255.04,Z 220.714,A -85,B 0,C 180,E1 -19854.052,E2 -19854.052} C_VEL
LIN {X 0,Y 257.577,Z 239.019,A -85,B 0,C 180,E1 -19855.251,E2 -19855.251} C_VEL
LIN {X 0,Y 255.113,Z 288.226,A -85,B 0,C 180,E1 -19856.684,E2 -19856.684} C_VEL
LIN {X 0,Y 253.615,Z 300.862,A -85,B 0,C 180,E1 -19857.291,E2 -19857.291} C_VEL
LIN {X 0,Y 251.461,Z 313.287,A -85,B 0,C 180,E1 -19858.161,E2 -19858.161} C_VEL
LIN {X 0,Y 248.97,Z 324.429,A -85,B 0,C 180,E1 -19859.227,E2 -19859.227} C_VEL
LIN {X 0,Y 245.848,Z 335.999,A -85,B 0,C 180,E1 -19860.689,E2 -19860.689} C_VEL
LIN {X 0,Y 242.748,Z 346.423,A -85,B 0,C 180,E1 -19862.404,E2 -19862.404} C_VEL
LIN {X 0,Y 239.495,Z 355.871,A -85,B 0,C 180,E1 -19864.352,E2 -19864.352} C_VEL
LIN {X 0,Y 236.003,Z 365.005,A -85,B 0,C 180,E1 -19866.76,E2 -19866.76} C_VEL
LIN {X 0,Y 233.089,Z 372.7,A -85,B 0,C 180,E1 -19869.378,E2 -19869.378} C_VEL
LIN {X 0,Y 230.465,Z 379.245,A -85,B 0,C 180,E1 -19872.245,E2 -19872.245} C_VEL
LIN {X 0,Y 228.511,Z 383.807,A -85,B 0,C 180,E1 -19874.845,E2 -19874.845} C_VEL
LIN {X 0,Y 227.136,Z 387.312,A -85,B 0,C 180,E1 -19877.491,E2 -19877.491} C_VEL
LIN {X 0,Y 226.048,Z 390.463,A -85,B 0,C 180,E1 -19881.057,E2 -19881.057} C_VEL
LIN {X 0,Y 225.65,Z 392.062,A -85,B 0,C 180,E1 -19884.638,E2 -19884.638} C_VEL
LIN {X 0,Y 225.686,Z 392.249,A -85,B 0,C 180,E1 -19886.429,E2 -19886.429} C_VEL
LIN {X 0,Y 225.829,Z 392.04,A -85,B 0,C 180,E1 -19888.216,E2 -19888.216} C_VEL
LIN {X 0,Y 225.881,Z 391.435,A -85,B 0,C 180,E1 -19890,E2 -19890} C_VEL
LIN {X 0,Y 225.857,Z 390.426,A -85,B 0,C 180,E1 -19891.783,E2 -19891.783} C_VEL
LIN {X 0,Y 225.746,Z 387.506,A -85,B 0,C 180,E1 -19894.969,E2 -19894.969} C_VEL
LIN {X 0,Y 225.924,Z 383.294,A -85,B 0,C 180,E1 -19898.047,E2 -19898.047} C_VEL
LIN {X 0,Y 226.396,Z 378.394,A -85,B 0,C 180,E1 -19900.734,E2 -19900.734} C_VEL
LIN {X 0,Y 227.244,Z 372.192,A -85,B 0,C 180,E1 -19903.412,E2 -19903.412} C_VEL
LIN {X 0,Y 228.498,Z 364.452,A -85,B 0,C 180,E1 -19906.07,E2 -19906.07} C_VEL
LIN {X 0,Y 229.681,Z 357.207,A -85,B 0,C 180,E1 -19908.089,E2 -19908.089} C_VEL
LIN {X 0,Y 231.473,Z 347.878,A -85,B 0,C 180,E1 -19910.204,E2 -19910.204} C_VEL
LIN {X 0,Y 233.238,Z 337.301,A -85,B 0,C 180,E1 -19912.126,E2 -19912.126} C_VEL
LIN {X 0,Y 234.811,Z 327.141,A -85,B 0,C 180,E1 -19913.598,E2 -19913.598} C_VEL
LIN {X 0,Y 236.5,Z 315.253,A -85,B 0,C 180,E1 -19914.936,E2 -19914.936} C_VEL
LIN {X 0,Y 237.929,Z 302.916,A -85,B 0,C 180,E1 -19915.946,E2 -19915.946} C_VEL
LIN {X 0,Y 238.886,Z 289.424,A -85,B 0,C 180,E1 -19916.704,E2 -19916.704} C_VEL
LIN {X 0,Y 240.22,Z 253.572,A -85,B 0,C 180,E1 -19917.809,E2 -19917.809} C_VEL
LIN {X 0,Y 240.72,Z 233.53,A -85,B 0,C 180,E1 -19918.415,E2 -19918.415} C_VEL
LIN {X 0,Y 236.007,Z 193.616,A -85,B 0,C 180,E1 -19920.208,E2 -19920.208} C_VEL
LIN {X 0,Y 230.964,Z 179.305,A -85,B 0,C 180,E1 -19921.278,E2 -19921.278} C_VEL
LIN {X 0,Y 228.845,Z 169.062,A -85,B 0,C 180,E1 -19925.274,E2 -19925.274} C_VEL
LIN {X 0,Y 227.939,Z 165.095,A -85,B 0,C 180,E1 -19926.941,E2 -19926.941} C_VEL
LIN {X 0,Y 227.834,Z 165.105,A -85,B 0,C 180,E1 -19930.374,E2 -19930.374} C_VEL
LIN {X 0,Y 227.834,Z 165.106,A -85,B 0,C 180,E1 -19935.192,E2 -19935.192} C_VEL
LIN {X 0,Y 227.826,Z 165.109,A -85,B 0,C 180,E1 -19939.623,E2 -19939.623} C_VEL
LIN {X 0,Y 227.884,Z 165.099,A -85,B 0,C 180,E1 -19944.128,E2 -19944.128} C_VEL
LIN {X 0,Y 227.872,Z 165.099,A -85,B 0,C 180,E1 -19948.378,E2 -19948.378} C_VEL
LIN {X 0,Y 227.887,Z 165.097,A -85,B 0,C 180,E1 -19952.445,E2 -19952.445} C_VEL
LIN {X 0,Y 227.907,Z 165.094,A -85,B 0,C 180,E1 -19956.366,E2 -19956.366} C_VEL
LIN {X 0,Y 227.923,Z 165.076,A -85,B 0,C 180,E1 -19960.172,E2 -19960.172} C_VEL
LIN {X 0,Y 228.023,Z 165.062,A -85,B 0,C 180,E1 -19963.895,E2 -19963.895} C_VEL
LIN {X 0,Y 228.056,Z 165.074,A -85,B 0,C 180,E1 -19967.542,E2 -19967.542} C_VEL
LIN {X 0,Y 228.253,Z 165.049,A -85,B 0,C 180,E1 -19971.144,E2 -19971.144} C_VEL
LIN {X 0,Y 228.303,Z 165.036,A -85,B 0,C 180,E1 -19972.927,E2 -19972.927} C_VEL
LIN {X 0,Y 228.553,Z 165.012,A -85,B 0,C 180,E1 -19978.238,E2 -19978.238} C_VEL
LIN {X 0,Y 228.554,Z 165.003,A -85,B 0,C 180,E1 -19981.762,E2 -19981.762} C_VEL
LIN {X 0,Y 228.324,Z 165.041,A -85,B 0,C 180,E1 -19987.072,E2 -19987.072} C_VEL
LIN {X 0,Y 228.145,Z 165.054,A -85,B 0,C 180,E1 -19990.651,E2 -19990.651} C_VEL
LIN {X 0,Y 228.064,Z 165.073,A -85,B 0,C 180,E1 -19994.272,E2 -19994.272} C_VEL
LIN {X 0,Y 228.002,Z 165.083,A -85,B 0,C 180,E1 -19997.953,E2 -19997.953} C_VEL
LIN {X 0,Y 227.916,Z 165.087,A -85,B 0,C 180,E1 -20002.321,E2 -20002.321} C_VEL
LIN {X 0,Y 227.941,Z 165.09,A -85,B 0,C 180,E1 -20006.602,E2 -20006.602} C_VEL
LIN {X 0,Y 227.896,Z 165.087,A -85,B 0,C 180,E1 -20010.291,E2 -20010.291} C_VEL
LIN {X 0,Y 227.877,Z 165.097,A -85,B 0,C 180,E1 -20013.72,E2 -20013.72} C_VEL
LIN {X 0,Y 227.844,Z 165.094,A -85,B 0,C 180,E1 -20018.091,E2 -20018.091} C_VEL
LIN {X 0,Y 227.81,Z 165.104,A -85,B 0,C 180,E1 -20022.742,E2 -20022.742} C_VEL
LIN {X 0,Y 227.81,Z 165.104,A -85,B 0,C 180,E1 -20027.258,E2 -20027.258} C_VEL
LIN {X 0,Y 227.843,Z 165.101,A -85,B 0,C 180,E1 -20031.909,E2 -20031.909} C_VEL
LIN {X 0,Y 227.878,Z 165.094,A -85,B 0,C 180,E1 -20036.377,E2 -20036.377} C_VEL
LIN {X 0,Y 227.918,Z 165.089,A -85,B 0,C 180,E1 -20040.438,E2 -20040.438} C_VEL
LIN {X 0,Y 227.924,Z 165.09,A -85,B 0,C 180,E1 -20044.426,E2 -20044.426} C_VEL
LIN {X 0,Y 227.944,Z 165.091,A -85,B 0,C 180,E1 -20048.286,E2 -20048.286} C_VEL
LIN {X 0,Y 228.008,Z 165.082,A -85,B 0,C 180,E1 -20052.848,E2 -20052.848} C_VEL
LIN {X 0,Y 228.057,Z 165.076,A -85,B 0,C 180,E1 -20057.543,E2 -20057.543} C_VEL
LIN {X 0,Y 228.131,Z 165.232,A -85,B 0,C 180,E1 -20058.671,E2 -20058.671} C_VEL
LIN {X 0,Y 229.185,Z 168.06,A -85,B 0,C 180,E1 -20058.896,E2 -20058.896} C_VEL
LIN {X 0,Y 235.453,Z 181.372,A -85,B 0,C 180,E1 -20060.065,E2 -20060.065} C_VEL
LIN {X 0,Y 241.739,Z 198.502,A -85,B 0,C 180,E1 -20061.29,E2 -20061.29} C_VEL
LIN {X 0,Y 239.351,Z 267.843,A -85,B 0,C 180,E1 -20063.361,E2 -20063.361} C_VEL
LIN {X 0,Y 238.501,Z 281.094,A -85,B 0,C 180,E1 -20064.081,E2 -20064.081} C_VEL
LIN {X 0,Y 237.435,Z 293.815,A -85,B 0,C 180,E1 -20065.119,E2 -20065.119} C_VEL
LIN {X 0,Y 236.1,Z 305.215,A -85,B 0,C 180,E1 -20066.374,E2 -20066.374} C_VEL
LIN {X 0,Y 234.384,Z 317.008,A -85,B 0,C 180,E1 -20068.067,E2 -20068.067} C_VEL
LIN {X 0,Y 232.714,Z 327.591,A -85,B 0,C 180,E1 -20070,E2 -20070} C_VEL
LIN {X 0,Y 230.954,Z 337.12,A -85,B 0,C 180,E1 -20072.18,E2 -20072.18} C_VEL
LIN {X 0,Y 229.515,Z 344.922,A -85,B 0,C 180,E1 -20074.391,E2 -20074.391} C_VEL
LIN {X 0,Y 228.152,Z 352.555,A -85,B 0,C 180,E1 -20077.078,E2 -20077.078} C_VEL
LIN {X 0,Y 227.123,Z 358.675,A -85,B 0,C 180,E1 -20079.799,E2 -20079.799} C_VEL
LIN {X 0,Y 226.377,Z 363.502,A -85,B 0,C 180,E1 -20082.552,E2 -20082.552} C_VEL
LIN {X 0,Y 225.854,Z 367.111,A -85,B 0,C 180,E1 -20085.283,E2 -20085.283} C_VEL
LIN {X 0,Y 225.564,Z 369.779,A -85,B 0,C 180,E1 -20088.154,E2 -20088.154} C_VEL
LIN {X 0,Y 225.599,Z 371.295,A -85,B 0,C 180,E1 -20090.841,E2 -20090.841} C_VEL
LIN {X 0,Y 225.882,Z 371.95,A -85,B 0,C 180,E1 -20093.859,E2 -20093.859} C_VEL
LIN {X 0,Y 226.28,Z 371.761,A -85,B 0,C 180,E1 -20095.774,E2 -20095.774} C_VEL
LIN {X 0,Y 226.821,Z 371.133,A -85,B 0,C 180,E1 -20097.696,E2 -20097.696} C_VEL
LIN {X 0,Y 227.825,Z 369.568,A -85,B 0,C 180,E1 -20100.26,E2 -20100.26} C_VEL
LIN {X 0,Y 229.549,Z 366.399,A -85,B 0,C 180,E1 -20103.443,E2 -20103.443} C_VEL
LIN {X 0,Y 231.541,Z 362.271,A -85,B 0,C 180,E1 -20106.291,E2 -20106.291} C_VEL
LIN {X 0,Y 234.043,Z 356.766,A -85,B 0,C 180,E1 -20109.095,E2 -20109.095} C_VEL
LIN {X 0,Y 236.827,Z 350.257,A -85,B 0,C 180,E1 -20111.637,E2 -20111.637} C_VEL
LIN {X 0,Y 239.915,Z 342.295,A -85,B 0,C 180,E1 -20114.086,E2 -20114.086} C_VEL
LIN {X 0,Y 243.147,Z 333.259,A -85,B 0,C 180,E1 -20116.271,E2 -20116.271} C_VEL
LIN {X 0,Y 246.332,Z 323.168,A -85,B 0,C 180,E1 -20118.177,E2 -20118.177} C_VEL
LIN {X 0,Y 249.377,Z 311.852,A -85,B 0,C 180,E1 -20119.858,E2 -20119.858} C_VEL
LIN {X 0,Y 251.845,Z 300.061,A -85,B 0,C 180,E1 -20121.227,E2 -20121.227} C_VEL
LIN {X 0,Y 253.929,Z 287.741,A -85,B 0,C 180,E1 -20122.275,E2 -20122.275} C_VEL
LIN {X 0,Y 255.49,Z 274.981,A -85,B 0,C 180,E1 -20123.041,E2 -20123.041} C_VEL
LIN {X 0,Y 256.492,Z 261.096,A -85,B 0,C 180,E1 -20123.544,E2 -20123.544} C_VEL
LIN {X 0,Y 258.756,Z 215.922,A -85,B 0,C 180,E1 -20124.797,E2 -20124.797} C_VEL
LIN {X 0,Y 252.504,Z 202.865,A -85,B 0,C 180,E1 -20126.603,E2 -20126.603} C_VEL
LIN {X 0,Y 247.724,Z 194.142,A -85,B 0,C 180,E1 -20128.031,E2 -20128.031} C_VEL
LIN {X 0,Y 240.768,Z 183.611,A -85,B 0,C 180,E1 -20130.189,E2 -20130.189} C_VEL
LIN {X 0,Y 237.148,Z 178.7,A -85,B 0,C 180,E1 -20131.393,E2 -20131.393} C_VEL
LIN {X 0,Y 234.391,Z 174.777,A -85,B 0,C 180,E1 -20132.367,E2 -20132.367} C_VEL
LIN {X 0,Y 232.085,Z 171.807,A -85,B 0,C 180,E1 -20133.2,E2 -20133.2} C_VEL
LIN {X 0,Y 231.417,Z 170.398,A -85,B 0,C 180,E1 -20133.475,E2 -20133.475} C_VEL
LIN {X 0,Y 229.085,Z 168.296,A -85,B 0,C 180,E1 -20134.314,E2 -20134.314} C_VEL
LIN {X 0,Y 227.988,Z 165.799,A -85,B 0,C 180,E1 -20134.8,E2 -20134.8} C_VEL
LIN {X 0,Y 227.873,Z 165.097,A -85,B 0,C 180,E1 -20134.908,E2 -20134.908} C_VEL
LIN {X 0,Y 227.919,Z 165.089,A -85,B 0,C 180,E1 -20138.283,E2 -20138.283} C_VEL
LIN {X 0,Y 227.999,Z 165.078,A -85,B 0,C 180,E1 -20143.894,E2 -20143.894} C_VEL
LIN {X 0,Y 228.125,Z 165.055,A -85,B 0,C 180,E1 -20149.348,E2 -20149.348} C_VEL
LIN {X 0,Y 228.305,Z 165.032,A -85,B 0,C 180,E1 -20152.927,E2 -20152.927} C_VEL
LIN {X 0,Y 228.533,Z 165.001,A -85,B 0,C 180,E1 -20158.238,E2 -20158.238} C_VEL
LIN {X 0,Y 228.535,Z 165.006,A -85,B 0,C 180,E1 -20161.763,E2 -20161.763} C_VEL
LIN {X 0,Y 228.302,Z 165.033,A -85,B 0,C 180,E1 -20167.073,E2 -20167.073} C_VEL
LIN {X 0,Y 228.144,Z 165.067,A -85,B 0,C 180,E1 -20170.652,E2 -20170.652} C_VEL
LIN {X 0,Y 228.043,Z 165.07,A -85,B 0,C 180,E1 -20174.274,E2 -20174.274} C_VEL
LIN {X 0,Y 227.972,Z 165.072,A -85,B 0,C 180,E1 -20177.956,E2 -20177.956} C_VEL
LIN {X 0,Y 227.922,Z 165.078,A -85,B 0,C 180,E1 -20182.323,E2 -20182.323} C_VEL
LIN {X 0,Y 227.876,Z 165.088,A -85,B 0,C 180,E1 -20184.06,E2 -20184.06} C_VEL
LIN {X 0,Y 227.176,Z 165.179,A -85,B 0,C 180,E1 -20185.534,E2 -20185.534} C_VEL
LIN {X 0,Y 224.3,Z 165.54,A -85,B 0,C 180,E1 -20187.94,E2 -20187.94} C_VEL
LIN {X 0,Y 221.883,Z 165.837,A -85,B 0,C 180,E1 -20189.902,E2 -20189.902} C_VEL
LIN {X 0,Y 220.861,Z 165.966,A -85,B 0,C 180,E1 -20191.427,E2 -20191.427} C_VEL
LIN {X 0,Y 220.785,Z 165.974,A -85,B 0,C 180,E1 -20191.943,E2 -20191.943} C_VEL
LIN {X 0,Y 220.859,Z 165.994,A -85,B 0,C 180,E1 -20196.88,E2 -20196.88} C_VEL
LIN {X 0,Y 222.816,Z 172.341,A -85,B 0,C 180,E1 -20201.482,E2 -20201.482} C_VEL
LIN {X 0,Y 224.048,Z 176.114,A -85,B 0,C 180,E1 -20203.844,E2 -20203.844} C_VEL
LIN {X 0,Y 227.018,Z 180.835,A -85,B 0,C 180,E1 -20205.086,E2 -20205.086} C_VEL
LIN {X 0,Y 228.464,Z 182.844,A -85,B 0,C 180,E1 -20205.652,E2 -20205.652} C_VEL
LIN {X 0,Y 232.37,Z 189.21,A -85,B 0,C 180,E1 -20207.159,E2 -20207.159} C_VEL
LIN {X 0,Y 235.729,Z 194.801,A -85,B 0,C 180,E1 -20208.385,E2 -20208.385} C_VEL
LIN {X 0,Y 240.042,Z 202.469,A -85,B 0,C 180,E1 -20209.876,E2 -20209.876} C_VEL
LIN {X 0,Y 245.985,Z 214.515,A -85,B 0,C 180,E1 -20211.83,E2 -20211.83} C_VEL
LIN {X 0,Y 250.052,Z 223.942,A -85,B 0,C 180,E1 -20213.125,E2 -20213.125} C_VEL
LIN {X 0,Y 252.231,Z 240.172,A -85,B 0,C 180,E1 -20214.23,E2 -20214.23} C_VEL
LIN {X 0,Y 249.724,Z 287.571,A -85,B 0,C 180,E1 -20215.629,E2 -20215.629} C_VEL
LIN {X 0,Y 248.174,Z 300.22,A -85,B 0,C 180,E1 -20216.237,E2 -20216.237} C_VEL
LIN {X 0,Y 245.973,Z 312.692,A -85,B 0,C 180,E1 -20217.12,E2 -20217.12} C_VEL
LIN {X 0,Y 243.364,Z 323.907,A -85,B 0,C 180,E1 -20218.194,E2 -20218.194} C_VEL
LIN {X 0,Y 240.13,Z 335.516,A -85,B 0,C 180,E1 -20219.677,E2 -20219.677} C_VEL
LIN {X 0,Y 236.845,Z 345.971,A -85,B 0,C 180,E1 -20221.413,E2 -20221.413} C_VEL
LIN {X 0,Y 233.804,Z 354.552,A -85,B 0,C 180,E1 -20223.199,E2 -20223.199} C_VEL
LIN {X 0,Y 230.647,Z 362.497,A -85,B 0,C 180,E1 -20225.23,E2 -20225.23} C_VEL
LIN {X 0,Y 227.425,Z 370.317,A -85,B 0,C 180,E1 -20227.755,E2 -20227.755} C_VEL
LIN {X 0,Y 225.262,Z 375.653,A -85,B 0,C 180,E1 -20229.928,E2 -20229.928} C_VEL
LIN {X 0,Y 222.991,Z 380.903,A -85,B 0,C 180,E1 -20232.577,E2 -20232.577} C_VEL
LIN {X 0,Y 221.05,Z 385.015,A -85,B 0,C 180,E1 -20235.265,E2 -20235.265} C_VEL
LIN {X 0,Y 220.158,Z 387.189,A -85,B 0,C 180,E1 -20237.087,E2 -20237.087} C_VEL
LIN {X 0,Y 219.013,Z 390.26,A -85,B 0,C 180,E1 -20240.767,E2 -20240.767} C_VEL
LIN {X 0,Y 218.692,Z 391.214,A -85,B 0,C 180,E1 -20242.614,E2 -20242.614} C_VEL
LIN {X 0,Y 218.596,Z 391.872,A -85,B 0,C 180,E1 -20245.328,E2 -20245.328} C_VEL
LIN {X 0,Y 218.756,Z 391.664,A -85,B 0,C 180,E1 -20248.159,E2 -20248.159} C_VEL
LIN {X 0,Y 218.812,Z 391.026,A -85,B 0,C 180,E1 -20250,E2 -20250} C_VEL
LIN {X 0,Y 218.764,Z 389.97,A -85,B 0,C 180,E1 -20251.841,E2 -20251.841} C_VEL
LIN {X 0,Y 218.655,Z 387.273,A -85,B 0,C 180,E1 -20254.856,E2 -20254.856} C_VEL
LIN {X 0,Y 218.773,Z 384.086,A -85,B 0,C 180,E1 -20257.382,E2 -20257.382} C_VEL
LIN {X 0,Y 219.18,Z 379.507,A -85,B 0,C 180,E1 -20260.157,E2 -20260.157} C_VEL
LIN {X 0,Y 220.107,Z 372.52,A -85,B 0,C 180,E1 -20263.385,E2 -20263.385} C_VEL
LIN {X 0,Y 221.395,Z 364.929,A -85,B 0,C 180,E1 -20266.126,E2 -20266.126} C_VEL
LIN {X 0,Y 222.505,Z 358.819,A -85,B 0,C 180,E1 -20267.936,E2 -20267.936} C_VEL
LIN {X 0,Y 223.407,Z 353.334,A -85,B 0,C 180,E1 -20269.352,E2 -20269.352} C_VEL
LIN {X 0,Y 225.319,Z 343.293,A -85,B 0,C 180,E1 -20271.499,E2 -20271.499} C_VEL
LIN {X 0,Y 227.043,Z 333.059,A -85,B 0,C 180,E1 -20273.245,E2 -20273.245} C_VEL
LIN {X 0,Y 228.814,Z 321.92,A -85,B 0,C 180,E1 -20274.739,E2 -20274.739} C_VEL
LIN {X 0,Y 230.458,Z 309.562,A -85,B 0,C 180,E1 -20276,E2 -20276} C_VEL
LIN {X 0,Y 231.76,Z 296.497,A -85,B 0,C 180,E1 -20276.934,E2 -20276.934} C_VEL
LIN {X 0,Y 232.576,Z 283.463,A -85,B 0,C 180,E1 -20277.527,E2 -20277.527} C_VEL
LIN {X 0,Y 234.11,Z 234.037,A -85,B 0,C 180,E1 -20279.045,E2 -20279.045} C_VEL
LIN {X 0,Y 229.679,Z 195.701,A -85,B 0,C 180,E1 -20280.825,E2 -20280.825} C_VEL
LIN {X 0,Y 223.679,Z 178.949,A -85,B 0,C 180,E1 -20282.148,E2 -20282.148} C_VEL
LIN {X 0,Y 221.741,Z 169.728,A -85,B 0,C 180,E1 -20285.897,E2 -20285.897} C_VEL
LIN {X 0,Y 220.871,Z 165.971,A -85,B 0,C 180,E1 -20287.534,E2 -20287.534} C_VEL
LIN {X 0,Y 220.776,Z 165.986,A -85,B 0,C 180,E1 -20291.951,E2 -20291.951} C_VEL
LIN {X 0,Y 220.774,Z 165.987,A -85,B 0,C 180,E1 -20295.546,E2 -20295.546} C_VEL
LIN {X 0,Y 220.807,Z 165.981,A -85,B 0,C 180,E1 -20300.463,E2 -20300.463} C_VEL
LIN {X 0,Y 220.804,Z 165.982,A -85,B 0,C 180,E1 -20305.045,E2 -20305.045} C_VEL
LIN {X 0,Y 220.869,Z 165.974,A -85,B 0,C 180,E1 -20309.394,E2 -20309.394} C_VEL
LIN {X 0,Y 220.895,Z 165.969,A -85,B 0,C 180,E1 -20313.549,E2 -20313.549} C_VEL
LIN {X 0,Y 220.864,Z 165.967,A -85,B 0,C 180,E1 -20317.552,E2 -20317.552} C_VEL
LIN {X 0,Y 220.924,Z 165.931,A -85,B 0,C 180,E1 -20322.621,E2 -20322.621} C_VEL
LIN {X 0,Y 220.995,Z 165.952,A -85,B 0,C 180,E1 -20327.137,E2 -20327.137} C_VEL
LIN {X 0,Y 221.194,Z 165.93,A -85,B 0,C 180,E1 -20330.859,E2 -20330.859} C_VEL
LIN {X 0,Y 221.127,Z 165.929,A -85,B 0,C 180,E1 -20334.528,E2 -20334.528} C_VEL
LIN {X 0,Y 221.511,Z 165.889,A -85,B 0,C 180,E1 -20338.181,E2 -20338.181} C_VEL
LIN {X 0,Y 221.512,Z 165.88,A -85,B 0,C 180,E1 -20341.818,E2 -20341.818} C_VEL
LIN {X 0,Y 221.259,Z 165.92,A -85,B 0,C 180,E1 -20347.299,E2 -20347.299} C_VEL
LIN {X 0,Y 221.067,Z 165.934,A -85,B 0,C 180,E1 -20350.996,E2 -20350.996} C_VEL
LIN {X 0,Y 220.996,Z 165.956,A -85,B 0,C 180,E1 -20354.738,E2 -20354.738} C_VEL
LIN {X 0,Y 220.92,Z 165.962,A -85,B 0,C 180,E1 -20358.549,E2 -20358.549} C_VEL
LIN {X 0,Y 220.884,Z 165.966,A -85,B 0,C 180,E1 -20362.675,E2 -20362.675} C_VEL
LIN {X 0,Y 220.882,Z 165.968,A -85,B 0,C 180,E1 -20367.014,E2 -20367.014} C_VEL
LIN {X 0,Y 220.837,Z 165.965,A -85,B 0,C 180,E1 -20370.767,E2 -20370.767} C_VEL
LIN {X 0,Y 220.801,Z 165.977,A -85,B 0,C 180,E1 -20374.955,E2 -20374.955} C_VEL
LIN {X 0,Y 220.805,Z 165.972,A -85,B 0,C 180,E1 -20379.537,E2 -20379.537} C_VEL
LIN {X 0,Y 220.772,Z 165.977,A -85,B 0,C 180,E1 -20384.454,E2 -20384.454} C_VEL
LIN {X 0,Y 220.769,Z 165.984,A -85,B 0,C 180,E1 -20388.048,E2 -20388.048} C_VEL
LIN {X 0,Y 220.823,Z 165.975,A -85,B 0,C 180,E1 -20392.793,E2 -20392.793} C_VEL
LIN {X 0,Y 220.817,Z 165.968,A -85,B 0,C 180,E1 -20397.244,E2 -20397.244} C_VEL
LIN {X 0,Y 220.836,Z 165.977,A -85,B 0,C 180,E1 -20401.487,E2 -20401.487} C_VEL
LIN {X 0,Y 220.861,Z 165.964,A -85,B 0,C 180,E1 -20405.565,E2 -20405.565} C_VEL
LIN {X 0,Y 220.875,Z 165.971,A -85,B 0,C 180,E1 -20409.513,E2 -20409.513} C_VEL
LIN {X 0,Y 220.99,Z 165.958,A -85,B 0,C 180,E1 -20413.369,E2 -20413.369} C_VEL
LIN {X 0,Y 221.033,Z 165.951,A -85,B 0,C 180,E1 -20417.799,E2 -20417.799} C_VEL
LIN {X 0,Y 222.157,Z 168.981,A -85,B 0,C 180,E1 -20418.073,E2 -20418.073} C_VEL
LIN {X 0,Y 229.009,Z 183.391,A -85,B 0,C 180,E1 -20419.415,E2 -20419.415} C_VEL
LIN {X 0,Y 232.382,Z 192.196,A -85,B 0,C 180,E1 -20420.099,E2 -20420.099} C_VEL
LIN {X 0,Y 235.26,Z 200.591,A -85,B 0,C 180,E1 -20420.695,E2 -20420.695} C_VEL
LIN {X 0,Y 232.7,Z 268.465,A -85,B 0,C 180,E1 -20422.767,E2 -20422.767} C_VEL
LIN {X 0,Y 231.828,Z 281.897,A -85,B 0,C 180,E1 -20423.527,E2 -20423.527} C_VEL
LIN {X 0,Y 230.653,Z 295.037,A -85,B 0,C 180,E1 -20424.646,E2 -20424.646} C_VEL
LIN {X 0,Y 229.109,Z 307.02,A -85,B 0,C 180,E1 -20426.043,E2 -20426.043} C_VEL
LIN {X 0,Y 227.353,Z 318.543,A -85,B 0,C 180,E1 -20427.786,E2 -20427.786} C_VEL
LIN {X 0,Y 225.665,Z 328.875,A -85,B 0,C 180,E1 -20429.777,E2 -20429.777} C_VEL
LIN {X 0,Y 224.052,Z 337.366,A -85,B 0,C 180,E1 -20431.798,E2 -20431.798} C_VEL
LIN {X 0,Y 222.533,Z 345.187,A -85,B 0,C 180,E1 -20434.075,E2 -20434.075} C_VEL
LIN {X 0,Y 221.13,Z 352.829,A -85,B 0,C 180,E1 -20436.845,E2 -20436.845} C_VEL
LIN {X 0,Y 220.215,Z 358.021,A -85,B 0,C 180,E1 -20439.182,E2 -20439.182} C_VEL
LIN {X 0,Y 219.389,Z 363.053,A -85,B 0,C 180,E1 -20442.019,E2 -20442.019} C_VEL
LIN {X 0,Y 218.817,Z 366.919,A -85,B 0,C 180,E1 -20444.889,E2 -20444.889} C_VEL
LIN {X 0,Y 218.572,Z 368.917,A -85,B 0,C 180,E1 -20446.822,E2 -20446.822} C_VEL
LIN {X 0,Y 218.44,Z 370.408,A -85,B 0,C 180,E1 -20448.768,E2 -20448.768} C_VEL
LIN {X 0,Y 218.528,Z 371.658,A -85,B 0,C 180,E1 -20451.148,E2 -20451.148} C_VEL
LIN {X 0,Y 218.925,Z 372.262,A -85,B 0,C 180,E1 -20454.667,E2 -20454.667} C_VEL
LIN {X 0,Y 219.42,Z 371.978,A -85,B 0,C 180,E1 -20456.643,E2 -20456.643} C_VEL
LIN {X 0,Y 220.029,Z 371.266,A -85,B 0,C 180,E1 -20458.628,E2 -20458.628} C_VEL
LIN {X 0,Y 220.994,Z 369.862,A -85,B 0,C 180,E1 -20460.836,E2 -20460.836} C_VEL
LIN {X 0,Y 222.474,Z 367.308,A -85,B 0,C 180,E1 -20463.562,E2 -20463.562} C_VEL
LIN {X 0,Y 224.525,Z 363.383,A -85,B 0,C 180,E1 -20466.494,E2 -20466.494} C_VEL
LIN {X 0,Y 227.016,Z 358.314,A -85,B 0,C 180,E1 -20469.29,E2 -20469.29} C_VEL
LIN {X 0,Y 229.641,Z 352.596,A -85,B 0,C 180,E1 -20471.732,E2 -20471.732} C_VEL
LIN {X 0,Y 232.515,Z 345.812,A -85,B 0,C 180,E1 -20474.043,E2 -20474.043} C_VEL
LIN {X 0,Y 235.528,Z 338.038,A -85,B 0,C 180,E1 -20476.171,E2 -20476.171} C_VEL
LIN {X 0,Y 238.991,Z 328.303,A -85,B 0,C 180,E1 -20478.263,E2 -20478.263} C_VEL
LIN {X 0,Y 242.065,Z 318.24,A -85,B 0,C 180,E1 -20479.976,E2 -20479.976} C_VEL
LIN {X 0,Y 244.842,Z 307.283,A -85,B 0,C 180,E1 -20481.462,E2 -20481.462} C_VEL
LIN {X 0,Y 247.078,Z 296.308,A -85,B 0,C 180,E1 -20482.624,E2 -20482.624} C_VEL
LIN {X 0,Y 249.088,Z 283.482,A -85,B 0,C 180,E1 -20483.615,E2 -20483.615} C_VEL
LIN {X 0,Y 250.496,Z 270.208,A -85,B 0,C 180,E1 -20484.306,E2 -20484.306} C_VEL
LIN {X 0,Y 253.325,Z 218.184,A -85,B 0,C 180,E1 -20485.82,E2 -20485.82} C_VEL
LIN {X 0,Y 246.81,Z 204.626,A -85,B 0,C 180,E1 -20487.807,E2 -20487.807} C_VEL
LIN {X 0,Y 242.733,Z 197.511,A -85,B 0,C 180,E1 -20489.082,E2 -20489.082} C_VEL
LIN {X 0,Y 236.646,Z 188.273,A -85,B 0,C 180,E1 -20491.084,E2 -20491.084} C_VEL
LIN {X 0,Y 230.933,Z 180.278,A -85,B 0,C 180,E1 -20493.127,E2 -20493.127} C_VEL
LIN {X 0,Y 228.344,Z 176.555,A -85,B 0,C 180,E1 -20494.124,E2 -20494.124} C_VEL
LIN {X 0,Y 225.475,Z 173.245,A -85,B 0,C 180,E1 -20495.239,E2 -20495.239} C_VEL
LIN {X 0,Y 224.365,Z 171.255,A -85,B 0,C 180,E1 -20495.725,E2 -20495.725} C_VEL
LIN {X 0,Y 222.068,Z 169.191,A -85,B 0,C 180,E1 -20496.652,E2 -20496.652} C_VEL
LIN {X 0,Y 220.965,Z 166.728,A -85,B 0,C 180,E1 -20497.205,E2 -20497.205} C_VEL
LIN {X 0,Y 220.839,Z 165.969,A -85,B 0,C 180,E1 -20497.354,E2 -20497.354} C_VEL
LIN {X 0,Y 220.863,Z 165.964,A -85,B 0,C 180,E1 -20501.446,E2 -20501.446} C_VEL
LIN {X 0,Y 220.92,Z 165.955,A -85,B 0,C 180,E1 -20505.256,E2 -20505.256} C_VEL
LIN {X 0,Y 221.196,Z 165.929,A -85,B 0,C 180,E1 -20510.859,E2 -20510.859} C_VEL
LIN {X 0,Y 221.243,Z 165.913,A -85,B 0,C 180,E1 -20512.7,E2 -20512.7} C_VEL
LIN {X 0,Y 221.466,Z 165.881,A -85,B 0,C 180,E1 -20518.182,E2 -20518.182} C_VEL
LIN {X 0,Y 221.469,Z 165.885,A -85,B 0,C 180,E1 -20521.819,E2 -20521.819} C_VEL
LIN {X 0,Y 221.24,Z 165.911,A -85,B 0,C 180,E1 -20527.3,E2 -20527.3} C_VEL
LIN {X 0,Y 221.065,Z 165.946,A -85,B 0,C 180,E1 -20530.997,E2 -20530.997} C_VEL
LIN {X 0,Y 220.994,Z 165.946,A -85,B 0,C 180,E1 -20536.632,E2 -20536.632} C_VEL
LIN {X 0,Y 220.882,Z 165.968,A -85,B 0,C 180,E1 -20540.487,E2 -20540.487} C_VEL
LIN {X 0,Y 220.85,Z 165.974,A -85,B 0,C 180,E1 -20544.437,E2 -20544.437} C_VEL
LIN {X 0,Y 220.806,Z 165.98,A -85,B 0,C 180,E1 -20548.518,E2 -20548.518} C_VEL
LIN {X 0,Y 220.785,Z 165.974,A -85,B 0,C 180,E1 -20551.943,E2 -20551.943} C_VEL
LIN {X 0,Y 220.245,Z 166.402,A -85,B 0,C 180,E1 -20553.461,E2 -20553.461} C_VEL
LIN {X 0,Y 218.977,Z 167.506,A -85,B 0,C 180,E1 -20554.945,E2 -20554.945} C_VEL
LIN {X 0,Y 216.274,Z 170.991,A -85,B 0,C 180,E1 -20557.878,E2 -20557.878} C_VEL
LIN {X 0,Y 215.845,Z 173.036,A -85,B 0,C 180,E1 -20559.364,E2 -20559.364} C_VEL
LIN {X 0,Y 215.97,Z 173.718,A -85,B 0,C 180,E1 -20559.859,E2 -20559.859} C_VEL
LIN {X 0,Y 216.543,Z 175.449,A -85,B 0,C 180,E1 -20561.011,E2 -20561.011} C_VEL
LIN {X 0,Y 219.852,Z 180.493,A -85,B 0,C 180,E1 -20562.597,E2 -20562.597} C_VEL
LIN {X 0,Y 221.361,Z 182.639,A -85,B 0,C 180,E1 -20563.267,E2 -20563.267} C_VEL
LIN {X 0,Y 224.537,Z 187.289,A -85,B 0,C 180,E1 -20564.612,E2 -20564.612} C_VEL
LIN {X 0,Y 229.334,Z 195.323,A -85,B 0,C 180,E1 -20566.554,E2 -20566.554} C_VEL
LIN {X 0,Y 233.951,Z 203.256,A -85,B 0,C 180,E1 -20568.288,E2 -20568.288} C_VEL
LIN {X 0,Y 240.382,Z 216.028,A -85,B 0,C 180,E1 -20570.557,E2 -20570.557} C_VEL
LIN {X 0,Y 245.118,Z 226.831,A -85,B 0,C 180,E1 -20572.143,E2 -20572.143} C_VEL
LIN {X 0,Y 246.983,Z 241.729,A -85,B 0,C 180,E1 -20573.175,E2 -20573.175} C_VEL
LIN {X 0,Y 244.444,Z 287.198,A -85,B 0,C 180,E1 -20574.533,E2 -20574.533} C_VEL
LIN {X 0,Y 242.847,Z 299.784,A -85,B 0,C 180,E1 -20575.14,E2 -20575.14} C_VEL
LIN {X 0,Y 240.508,Z 312.302,A -85,B 0,C 180,E1 -20576.023,E2 -20576.023} C_VEL
LIN {X 0,Y 237.842,Z 323.509,A -85,B 0,C 180,E1 -20577.114,E2 -20577.114} C_VEL
LIN {X 0,Y 234.496,Z 335.109,A -85,B 0,C 180,E1 -20578.618,E2 -20578.618} C_VEL
LIN {X 0,Y 231.069,Z 345.557,A -85,B 0,C 180,E1 -20580.38,E2 -20580.38} C_VEL
LIN {X 0,Y 227.51,Z 355.024,A -85,B 0,C 180,E1 -20582.395,E2 -20582.395} C_VEL
LIN {X 0,Y 223.631,Z 364.188,A -85,B 0,C 180,E1 -20584.896,E2 -20584.896} C_VEL
LIN {X 0,Y 220.378,Z 371.602,A -85,B 0,C 180,E1 -20587.499,E2 -20587.499} C_VEL
LIN {X 0,Y 217.734,Z 377.59,A -85,B 0,C 180,E1 -20590.189,E2 -20590.189} C_VEL
LIN {X 0,Y 215.487,Z 382.361,A -85,B 0,C 180,E1 -20592.93,E2 -20592.93} C_VEL
LIN {X 0,Y 213.659,Z 386.048,A -85,B 0,C 180,E1 -20595.717,E2 -20595.717} C_VEL
LIN {X 0,Y 212.506,Z 388.755,A -85,B 0,C 180,E1 -20598.554,E2 -20598.554} C_VEL
LIN {X 0,Y 211.631,Z 390.969,A -85,B 0,C 180,E1 -20602.366,E2 -20602.366} C_VEL
LIN {X 0,Y 211.502,Z 391.561,A -85,B 0,C 180,E1 -20606.189,E2 -20606.189} C_VEL
LIN {X 0,Y 211.661,Z 391.285,A -85,B 0,C 180,E1 -20608.097,E2 -20608.097} C_VEL
LIN {X 0,Y 211.744,Z 390.612,A -85,B 0,C 180,E1 -20610,E2 -20610} C_VEL
LIN {X 0,Y 211.673,Z 389.486,A -85,B 0,C 180,E1 -20611.902,E2 -20611.902} C_VEL
LIN {X 0,Y 211.566,Z 387.02,A -85,B 0,C 180,E1 -20614.742,E2 -20614.742} C_VEL
LIN {X 0,Y 211.696,Z 383.462,A -85,B 0,C 180,E1 -20617.631,E2 -20617.631} C_VEL
LIN {X 0,Y 212.137,Z 378.786,A -85,B 0,C 180,E1 -20620.498,E2 -20620.498} C_VEL
LIN {X 0,Y 213.169,Z 371.692,A -85,B 0,C 180,E1 -20623.829,E2 -20623.829} C_VEL
LIN {X 0,Y 214.506,Z 363.986,A -85,B 0,C 180,E1 -20626.659,E2 -20626.659} C_VEL
LIN {X 0,Y 215.621,Z 357.745,A -85,B 0,C 180,E1 -20628.529,E2 -20628.529} C_VEL
LIN {X 0,Y 217.474,Z 348.526,A -85,B 0,C 180,E1 -20630.823,E2 -20630.823} C_VEL
LIN {X 0,Y 219.365,Z 338.271,A -85,B 0,C 180,E1 -20632.858,E2 -20632.858} C_VEL
LIN {X 0,Y 221.013,Z 328.463,A -85,B 0,C 180,E1 -20634.417,E2 -20634.417} C_VEL
LIN {X 0,Y 222.914,Z 316.067,A -85,B 0,C 180,E1 -20635.941,E2 -20635.941} C_VEL
LIN {X 0,Y 224.371,Z 304.345,A -85,B 0,C 180,E1 -20637.012,E2 -20637.012} C_VEL
LIN {X 0,Y 225.452,Z 291.805,A -85,B 0,C 180,E1 -20637.815,E2 -20637.815} C_VEL
LIN {X 0,Y 226.232,Z 275.66,A -85,B 0,C 180,E1 -20638.418,E2 -20638.418} C_VEL
LIN {X 0,Y 227.506,Z 234.381,A -85,B 0,C 180,E1 -20639.719,E2 -20639.719} C_VEL
LIN {X 0,Y 223.311,Z 197.548,A -85,B 0,C 180,E1 -20641.494,E2 -20641.494} C_VEL
LIN {X 0,Y 216.377,Z 178.555,A -85,B 0,C 180,E1 -20643.104,E2 -20643.104} C_VEL
LIN {X 0,Y 214.57,Z 170.145,A -85,B 0,C 180,E1 -20646.658,E2 -20646.658} C_VEL
LIN {X 0,Y 213.812,Z 166.85,A -85,B 0,C 180,E1 -20648.203,E2 -20648.203} C_VEL
LIN {X 0,Y 213.717,Z 166.864,A -85,B 0,C 180,E1 -20651.124,E2 -20651.124} C_VEL
LIN {X 0,Y 213.708,Z 166.867,A -85,B 0,C 180,E1 -20653.678,E2 -20653.678} C_VEL
LIN {X 0,Y 213.706,Z 166.866,A -85,B 0,C 180,E1 -20656.343,E2 -20656.343} C_VEL
LIN {X 0,Y 213.718,Z 166.866,A -85,B 0,C 180,E1 -20659.142,E2 -20659.142} C_VEL
LIN {X 0,Y 213.745,Z 166.863,A -85,B 0,C 180,E1 -20663.711,E2 -20663.711} C_VEL
LIN {X 0,Y 213.796,Z 166.853,A -85,B 0,C 180,E1 -20668.724,E2 -20668.724} C_VEL
LIN {X 0,Y 213.826,Z 166.849,A -85,B 0,C 180,E1 -20672.603,E2 -20672.603} C_VEL
LIN {X 0,Y 213.819,Z 166.849,A -85,B 0,C 180,E1 -20676.973,E2 -20676.973} C_VEL
LIN {X 0,Y 213.888,Z 166.807,A -85,B 0,C 180,E1 -20682.799,E2 -20682.799} C_VEL
LIN {X 0,Y 213.935,Z 166.828,A -85,B 0,C 180,E1 -20686.705,E2 -20686.705} C_VEL
LIN {X 0,Y 214.134,Z 166.81,A -85,B 0,C 180,E1 -20690.554,E2 -20690.554} C_VEL
LIN {X 0,Y 214.088,Z 166.804,A -85,B 0,C 180,E1 -20694.348,E2 -20694.348} C_VEL
LIN {X 0,Y 214.443,Z 166.769,A -85,B 0,C 180,E1 -20698.122,E2 -20698.122} C_VEL
LIN {X 0,Y 214.55,Z 166.754,A -85,B 0,C 180,E1 -20700,E2 -20700} C_VEL
LIN {X 0,Y 214.445,Z 166.76,A -85,B 0,C 180,E1 -20701.878,E2 -20701.878} C_VEL
LIN {X 0,Y 214.198,Z 166.799,A -85,B 0,C 180,E1 -20707.541,E2 -20707.541} C_VEL
LIN {X 0,Y 213.999,Z 166.812,A -85,B 0,C 180,E1 -20711.364,E2 -20711.364} C_VEL
LIN {X 0,Y 213.933,Z 166.834,A -85,B 0,C 180,E1 -20715.237,E2 -20715.237} C_VEL
LIN {X 0,Y 213.835,Z 166.842,A -85,B 0,C 180,E1 -20719.187,E2 -20719.187} C_VEL
LIN {X 0,Y 213.81,Z 166.846,A -85,B 0,C 180,E1 -20723.231,E2 -20723.231} C_VEL
LIN {X 0,Y 213.828,Z 166.847,A -85,B 0,C 180,E1 -20727.45,E2 -20727.45} C_VEL
LIN {X 0,Y 213.766,Z 166.848,A -85,B 0,C 180,E1 -20731.737,E2 -20731.737} C_VEL
LIN {X 0,Y 213.743,Z 166.854,A -85,B 0,C 180,E1 -20736.288,E2 -20736.288} C_VEL
LIN {X 0,Y 213.711,Z 166.86,A -85,B 0,C 180,E1 -20741.125,E2 -20741.125} C_VEL
LIN {X 0,Y 213.705,Z 166.861,A -85,B 0,C 180,E1 -20743.678,E2 -20743.678} C_VEL
LIN {X 0,Y 213.705,Z 166.86,A -85,B 0,C 180,E1 -20746.344,E2 -20746.344} C_VEL
LIN {X 0,Y 213.716,Z 166.863,A -85,B 0,C 180,E1 -20749.143,E2 -20749.143} C_VEL
LIN {X 0,Y 213.743,Z 166.861,A -85,B 0,C 180,E1 -20753.712,E2 -20753.712} C_VEL
LIN {X 0,Y 213.794,Z 166.837,A -85,B 0,C 180,E1 -20758.725,E2 -20758.725} C_VEL
LIN {X 0,Y 213.825,Z 166.85,A -85,B 0,C 180,E1 -20762.604,E2 -20762.604} C_VEL
LIN {X 0,Y 213.818,Z 166.845,A -85,B 0,C 180,E1 -20766.974,E2 -20766.974} C_VEL
LIN {X 0,Y 213.921,Z 166.837,A -85,B 0,C 180,E1 -20772.802,E2 -20772.802} C_VEL
LIN {X 0,Y 213.933,Z 166.839,A -85,B 0,C 180,E1 -20776.876,E2 -20776.876} C_VEL
LIN {X 0,Y 214.963,Z 169.673,A -85,B 0,C 180,E1 -20777.168,E2 -20777.168} C_VEL
LIN {X 0,Y 222.714,Z 185.612,A -85,B 0,C 180,E1 -20778.748,E2 -20778.748} C_VEL
LIN {X 0,Y 226.353,Z 195.148,A -85,B 0,C 180,E1 -20779.522,E2 -20779.522} C_VEL
LIN {X 0,Y 228.695,Z 202.157,A -85,B 0,C 180,E1 -20780.035,E2 -20780.035} C_VEL
LIN {X 0,Y 226.107,Z 268.856,A -85,B 0,C 180,E1 -20782.128,E2 -20782.128} C_VEL
LIN {X 0,Y 225.169,Z 282.708,A -85,B 0,C 180,E1 -20782.941,E2 -20782.941} C_VEL
LIN {X 0,Y 223.995,Z 295.177,A -85,B 0,C 180,E1 -20784.035,E2 -20784.035} C_VEL
LIN {X 0,Y 222.407,Z 307.196,A -85,B 0,C 180,E1 -20785.469,E2 -20785.469} C_VEL
LIN {X 0,Y 220.587,Z 318.745,A -85,B 0,C 180,E1 -20787.261,E2 -20787.261} C_VEL
LIN {X 0,Y 218.821,Z 329.109,A -85,B 0,C 180,E1 -20789.31,E2 -20789.31} C_VEL
LIN {X 0,Y 216.792,Z 339.29,A -85,B 0,C 180,E1 -20791.858,E2 -20791.858} C_VEL
LIN {X 0,Y 215.074,Z 348.207,A -85,B 0,C 180,E1 -20794.686,E2 -20794.686} C_VEL
LIN {X 0,Y 213.721,Z 355.302,A -85,B 0,C 180,E1 -20797.559,E2 -20797.559} C_VEL
LIN {X 0,Y 212.686,Z 360.982,A -85,B 0,C 180,E1 -20800.472,E2 -20800.472} C_VEL
LIN {X 0,Y 211.994,Z 365.423,A -85,B 0,C 180,E1 -20803.419,E2 -20803.419} C_VEL
LIN {X 0,Y 211.614,Z 367.992,A -85,B 0,C 180,E1 -20805.608,E2 -20805.608} C_VEL
LIN {X 0,Y 211.419,Z 369.629,A -85,B 0,C 180,E1 -20807.409,E2 -20807.409} C_VEL
LIN {X 0,Y 211.365,Z 371.029,A -85,B 0,C 180,E1 -20809.421,E2 -20809.421} C_VEL
LIN {X 0,Y 211.453,Z 372.016,A -85,B 0,C 180,E1 -20811.468,E2 -20811.468} C_VEL
LIN {X 0,Y 211.638,Z 372.502,A -85,B 0,C 180,E1 -20813.484,E2 -20813.484} C_VEL
LIN {X 0,Y 212.307,Z 372.407,A -85,B 0,C 180,E1 -20816.648,E2 -20816.648} C_VEL
LIN {X 0,Y 213.296,Z 371.33,A -85,B 0,C 180,E1 -20819.62,E2 -20819.62} C_VEL
LIN {X 0,Y 214.273,Z 370.006,A -85,B 0,C 180,E1 -20821.654,E2 -20821.654} C_VEL
LIN {X 0,Y 216.046,Z 367.095,A -85,B 0,C 180,E1 -20824.7,E2 -20824.7} C_VEL
LIN {X 0,Y 218.31,Z 362.978,A -85,B 0,C 180,E1 -20827.71,E2 -20827.71} C_VEL
LIN {X 0,Y 221.268,Z 357.215,A -85,B 0,C 180,E1 -20830.781,E2 -20830.781} C_VEL
LIN {X 0,Y 224.511,Z 350.417,A -85,B 0,C 180,E1 -20833.526,E2 -20833.526} C_VEL
LIN {X 0,Y 227.652,Z 343.081,A -85,B 0,C 180,E1 -20835.871,E2 -20835.871} C_VEL
LIN {X 0,Y 230.906,Z 334.858,A -85,B 0,C 180,E1 -20837.964,E2 -20837.964} C_VEL
LIN {X 0,Y 234.304,Z 325.301,A -85,B 0,C 180,E1 -20839.897,E2 -20839.897} C_VEL
LIN {X 0,Y 237.498,Z 314.711,A -85,B 0,C 180,E1 -20841.58,E2 -20841.58} C_VEL
LIN {X 0,Y 240.471,Z 302.248,A -85,B 0,C 180,E1 -20843.137,E2 -20843.137} C_VEL
LIN {X 0,Y 242.876,Z 289.7,A -85,B 0,C 180,E1 -20844.272,E2 -20844.272} C_VEL
LIN {X 0,Y 244.623,Z 276.915,A -85,B 0,C 180,E1 -20845.089,E2 -20845.089} C_VEL
LIN {X 0,Y 245.656,Z 264.61,A -85,B 0,C 180,E1 -20845.596,E2 -20845.596} C_VEL
LIN {X 0,Y 248.096,Z 220.747,A -85,B 0,C 180,E1 -20846.849,E2 -20846.849} C_VEL
LIN {X 0,Y 241.562,Z 207.119,A -85,B 0,C 180,E1 -20848.954,E2 -20848.954} C_VEL
LIN {X 0,Y 235.632,Z 197.424,A -85,B 0,C 180,E1 -20850.937,E2 -20850.937} C_VEL
LIN {X 0,Y 230.002,Z 189.207,A -85,B 0,C 180,E1 -20852.964,E2 -20852.964} C_VEL
LIN {X 0,Y 227.201,Z 185.334,A -85,B 0,C 180,E1 -20854.035,E2 -20854.035} C_VEL
LIN {X 0,Y 224.553,Z 181.663,A -85,B 0,C 180,E1 -20855.097,E2 -20855.097} C_VEL
LIN {X 0,Y 221.966,Z 178.186,A -85,B 0,C 180,E1 -20856.18,E2 -20856.18} C_VEL
LIN {X 0,Y 221.003,Z 177.016,A -85,B 0,C 180,E1 -20856.596,E2 -20856.596} C_VEL
LIN {X 0,Y 218.626,Z 174.153,A -85,B 0,C 180,E1 -20857.662,E2 -20857.662} C_VEL
LIN {X 0,Y 217.561,Z 172.275,A -85,B 0,C 180,E1 -20858.193,E2 -20858.193} C_VEL
LIN {X 0,Y 215.128,Z 170.195,A -85,B 0,C 180,E1 -20859.315,E2 -20859.315} C_VEL
LIN {X 0,Y 213.989,Z 167.82,A -85,B 0,C 180,E1 -20859.953,E2 -20859.953} C_VEL
LIN {X 0,Y 213.789,Z 166.848,A -85,B 0,C 180,E1 -20860.184,E2 -20860.184} C_VEL
LIN {X 0,Y 213.879,Z 166.844,A -85,B 0,C 180,E1 -20862.799,E2 -20862.799} C_VEL
LIN {X 0,Y 213.909,Z 166.839,A -85,B 0,C 180,E1 -20866.704,E2 -20866.704} C_VEL
LIN {X 0,Y 214.135,Z 166.805,A -85,B 0,C 180,E1 -20870.555,E2 -20870.555} C_VEL
LIN {X 0,Y 214.072,Z 166.805,A -85,B 0,C 180,E1 -20874.348,E2 -20874.348} C_VEL
LIN {X 0,Y 214.403,Z 166.76,A -85,B 0,C 180,E1 -20878.122,E2 -20878.122} C_VEL
LIN {X 0,Y 214.513,Z 166.759,A -85,B 0,C 180,E1 -20880,E2 -20880} C_VEL
LIN {X 0,Y 214.406,Z 166.764,A -85,B 0,C 180,E1 -20881.879,E2 -20881.879} C_VEL
LIN {X 0,Y 214.182,Z 166.789,A -85,B 0,C 180,E1 -20887.542,E2 -20887.542} C_VEL
LIN {X 0,Y 213.996,Z 166.821,A -85,B 0,C 180,E1 -20891.365,E2 -20891.365} C_VEL
LIN {X 0,Y 213.912,Z 166.839,A -85,B 0,C 180,E1 -20895.239,E2 -20895.239} C_VEL
LIN {X 0,Y 213.824,Z 166.842,A -85,B 0,C 180,E1 -20899.189,E2 -20899.189} C_VEL
LIN {X 0,Y 213.805,Z 166.839,A -85,B 0,C 180,E1 -20903.232,E2 -20903.232} C_VEL
LIN {X 0,Y 213.789,Z 166.843,A -85,B 0,C 180,E1 -20907.428,E2 -20907.428} C_VEL
LIN {X 0,Y 213.749,Z 166.852,A -85,B 0,C 180,E1 -20911.913,E2 -20911.913} C_VEL
LIN {X 0,Y 213.783,Z 166.889,A -85,B 0,C 180,E1 -20914.408,E2 -20914.408} C_VEL
LIN {X 0,Y 215.97,Z 173.718,A -85,B 0,C 180,E1 -20919.859,E2 -20919.859} C_VEL
LIN {X 0,Y 216.584,Z 175.501,A -85,B 0,C 180,E1 -20920.748,E2 -20920.748} C_VEL
LIN {X 0,Y 218.016,Z 179.408,A -85,B 0,C 180,E1 -20921.828,E2 -20921.828} C_VEL
LIN {X 0,Y 219.55,Z 184.093,A -85,B 0,C 180,E1 -20922.693,E2 -20922.693} C_VEL
LIN {X 0,Y 222.607,Z 194.233,A -85,B 0,C 180,E1 -20924.333,E2 -20924.333} C_VEL
LIN {X 0,Y 223.955,Z 197.26,A -85,B 0,C 180,E1 -20924.95,E2 -20924.95} C_VEL
LIN {X 0,Y 230.109,Z 208.066,A -85,B 0,C 180,E1 -20927.417,E2 -20927.417} C_VEL
LIN {X 0,Y 236.091,Z 220.255,A -85,B 0,C 180,E1 -20929.659,E2 -20929.659} C_VEL
LIN {X 0,Y 240.342,Z 230.476,A -85,B 0,C 180,E1 -20931.175,E2 -20931.175} C_VEL
LIN {X 0,Y 241.803,Z 242.701,A -85,B 0,C 180,E1 -20932.045,E2 -20932.045} C_VEL
LIN {X 0,Y 239.218,Z 286.848,A -85,B 0,C 180,E1 -20933.38,E2 -20933.38} C_VEL
LIN {X 0,Y 237.475,Z 300.105,A -85,B 0,C 180,E1 -20934.036,E2 -20934.036} C_VEL
LIN {X 0,Y 234.95,Z 312.977,A -85,B 0,C 180,E1 -20934.973,E2 -20934.973} C_VEL
LIN {X 0,Y 231.968,Z 324.701,A -85,B 0,C 180,E1 -20936.171,E2 -20936.171} C_VEL
LIN {X 0,Y 228.511,Z 336.019,A -85,B 0,C 180,E1 -20937.698,E2 -20937.698} C_VEL
LIN {X 0,Y 224.97,Z 346.256,A -85,B 0,C 180,E1 -20939.492,E2 -20939.492} C_VEL
LIN {X 0,Y 221.273,Z 355.505,A -85,B 0,C 180,E1 -20941.547,E2 -20941.547} C_VEL
LIN {X 0,Y 217.223,Z 364.51,A -85,B 0,C 180,E1 -20944.101,E2 -20944.101} C_VEL
LIN {X 0,Y 213.837,Z 371.795,A -85,B 0,C 180,E1 -20946.771,E2 -20946.771} C_VEL
LIN {X 0,Y 211.062,Z 377.672,A -85,B 0,C 180,E1 -20949.535,E2 -20949.535} C_VEL
LIN {X 0,Y 208.708,Z 382.348,A -85,B 0,C 180,E1 -20952.358,E2 -20952.358} C_VEL
LIN {X 0,Y 206.775,Z 385.956,A -85,B 0,C 180,E1 -20955.231,E2 -20955.231} C_VEL
LIN {X 0,Y 205.512,Z 388.588,A -85,B 0,C 180,E1 -20958.159,E2 -20958.159} C_VEL
LIN {X 0,Y 204.959,Z 389.855,A -85,B 0,C 180,E1 -20960.128,E2 -20960.128} C_VEL
LIN {X 0,Y 204.592,Z 390.701,A -85,B 0,C 180,E1 -20962.102,E2 -20962.102} C_VEL
LIN {X 0,Y 204.426,Z 391.218,A -85,B 0,C 180,E1 -20966.057,E2 -20966.057} C_VEL
LIN {X 0,Y 204.568,Z 390.905,A -85,B 0,C 180,E1 -20968.031,E2 -20968.031} C_VEL
LIN {X 0,Y 204.678,Z 390.184,A -85,B 0,C 180,E1 -20970,E2 -20970} C_VEL
LIN {X 0,Y 204.584,Z 388.999,A -85,B 0,C 180,E1 -20971.968,E2 -20971.968} C_VEL
LIN {X 0,Y 204.503,Z 386.676,A -85,B 0,C 180,E1 -20974.705,E2 -20974.705} C_VEL
LIN {X 0,Y 204.64,Z 382.818,A -85,B 0,C 180,E1 -20977.895,E2 -20977.895} C_VEL
LIN {X 0,Y 205.11,Z 378.051,A -85,B 0,C 180,E1 -20980.862,E2 -20980.862} C_VEL
LIN {X 0,Y 206.222,Z 370.862,A -85,B 0,C 180,E1 -20984.304,E2 -20984.304} C_VEL
LIN {X 0,Y 207.663,Z 363.005,A -85,B 0,C 180,E1 -20987.225,E2 -20987.225} C_VEL
LIN {X 0,Y 208.772,Z 356.672,A -85,B 0,C 180,E1 -20989.16,E2 -20989.16} C_VEL
LIN {X 0,Y 210.831,Z 347.287,A -85,B 0,C 180,E1 -20991.511,E2 -20991.511} C_VEL
LIN {X 0,Y 212.786,Z 336.78,A -85,B 0,C 180,E1 -20993.607,E2 -20993.607} C_VEL
LIN {X 0,Y 214.509,Z 326.709,A -85,B 0,C 180,E1 -20995.209,E2 -20995.209} C_VEL
LIN {X 0,Y 216.341,Z 314.947,A -85,B 0,C 180,E1 -20996.661,E2 -20996.661} C_VEL
LIN {X 0,Y 217.981,Z 302.184,A -85,B 0,C 180,E1 -20997.806,E2 -20997.806} C_VEL
LIN {X 0,Y 219.068,Z 288.569,A -85,B 0,C 180,E1 -20998.634,E2 -20998.634} C_VEL
LIN {X 0,Y 220.59,Z 251.439,A -85,B 0,C 180,E1 -20999.871,E2 -20999.871} C_VEL
LIN {X 0,Y 220.961,Z 234.92,A -85,B 0,C 180,E1 -21000.424,E2 -21000.424} C_VEL
LIN {X 0,Y 216.918,Z 199.349,A -85,B 0,C 180,E1 -21002.211,E2 -21002.211} C_VEL
LIN {X 0,Y 210.308,Z 181.504,A -85,B 0,C 180,E1 -21003.754,E2 -21003.754} C_VEL
LIN {X 0,Y 209.099,Z 178.166,A -85,B 0,C 180,E1 -21004.111,E2 -21004.111} C_VEL
LIN {X 0,Y 207.149,Z 169.488,A -85,B 0,C 180,E1 -21007.962,E2 -21007.962} C_VEL
LIN {X 0,Y 206.74,Z 167.733,A -85,B 0,C 180,E1 -21008.861,E2 -21008.861} C_VEL
LIN {X 0,Y 206.627,Z 167.747,A -85,B 0,C 180,E1 -21012.863,E2 -21012.863} C_VEL
LIN {X 0,Y 206.625,Z 167.749,A -85,B 0,C 180,E1 -21017.135,E2 -21017.135} C_VEL
LIN {X 0,Y 206.689,Z 167.742,A -85,B 0,C 180,E1 -21021.449,E2 -21021.449} C_VEL
LIN {X 0,Y 206.699,Z 167.738,A -85,B 0,C 180,E1 -21024.688,E2 -21024.688} C_VEL
LIN {X 0,Y 206.724,Z 167.736,A -85,B 0,C 180,E1 -21029.339,E2 -21029.339} C_VEL
LIN {X 0,Y 206.732,Z 167.733,A -85,B 0,C 180,E1 -21033.771,E2 -21033.771} C_VEL
LIN {X 0,Y 206.735,Z 167.725,A -85,B 0,C 180,E1 -21038.04,E2 -21038.04} C_VEL
LIN {X 0,Y 206.821,Z 167.683,A -85,B 0,C 180,E1 -21042.192,E2 -21042.192} C_VEL
LIN {X 0,Y 206.876,Z 167.705,A -85,B 0,C 180,E1 -21046.243,E2 -21046.243} C_VEL
LIN {X 0,Y 207.079,Z 167.688,A -85,B 0,C 180,E1 -21050.23,E2 -21050.23} C_VEL
LIN {X 0,Y 207.049,Z 167.68,A -85,B 0,C 180,E1 -21054.155,E2 -21054.155} C_VEL
LIN {X 0,Y 207.38,Z 167.649,A -85,B 0,C 180,E1 -21058.058,E2 -21058.058} C_VEL
LIN {X 0,Y 207.515,Z 167.63,A -85,B 0,C 180,E1 -21060,E2 -21060} C_VEL
LIN {X 0,Y 207.382,Z 167.639,A -85,B 0,C 180,E1 -21061.942,E2 -21061.942} C_VEL
LIN {X 0,Y 207.141,Z 167.679,A -85,B 0,C 180,E1 -21067.8,E2 -21067.8} C_VEL
LIN {X 0,Y 206.924,Z 167.693,A -85,B 0,C 180,E1 -21071.758,E2 -21071.758} C_VEL
LIN {X 0,Y 206.867,Z 167.715,A -85,B 0,C 180,E1 -21075.77,E2 -21075.77} C_VEL
LIN {X 0,Y 206.778,Z 167.719,A -85,B 0,C 180,E1 -21079.869,E2 -21079.869} C_VEL
LIN {X 0,Y 206.746,Z 167.729,A -85,B 0,C 180,E1 -21084.074,E2 -21084.074} C_VEL
LIN {X 0,Y 206.736,Z 167.726,A -85,B 0,C 180,E1 -21088.42,E2 -21088.42} C_VEL
LIN {X 0,Y 206.698,Z 167.732,A -85,B 0,C 180,E1 -21092.957,E2 -21092.957} C_VEL
LIN {X 0,Y 206.679,Z 167.729,A -85,B 0,C 180,E1 -21097.74,E2 -21097.74} C_VEL
LIN {X 0,Y 206.641,Z 167.742,A -85,B 0,C 180,E1 -21101.563,E2 -21101.563} C_VEL
LIN {X 0,Y 206.632,Z 167.737,A -85,B 0,C 180,E1 -21105.582,E2 -21105.582} C_VEL
LIN {X 0,Y 206.659,Z 167.74,A -85,B 0,C 180,E1 -21109.749,E2 -21109.749} C_VEL
LIN {X 0,Y 206.698,Z 167.737,A -85,B 0,C 180,E1 -21114.689,E2 -21114.689} C_VEL
LIN {X 0,Y 206.722,Z 167.719,A -85,B 0,C 180,E1 -21119.339,E2 -21119.339} C_VEL
LIN {X 0,Y 206.73,Z 167.731,A -85,B 0,C 180,E1 -21123.772,E2 -21123.772} C_VEL
LIN {X 0,Y 206.735,Z 167.734,A -85,B 0,C 180,E1 -21128.041,E2 -21128.041} C_VEL
LIN {X 0,Y 206.867,Z 167.713,A -85,B 0,C 180,E1 -21132.196,E2 -21132.196} C_VEL
LIN {X 0,Y 206.862,Z 167.782,A -85,B 0,C 180,E1 -21135.968,E2 -21135.968} C_VEL
LIN {X 0,Y 207.962,Z 170.699,A -85,B 0,C 180,E1 -21136.242,E2 -21136.242} C_VEL
LIN {X 0,Y 216.51,Z 188.089,A -85,B 0,C 180,E1 -21138.06,E2 -21138.06} C_VEL
LIN {X 0,Y 219.866,Z 196.657,A -85,B 0,C 180,E1 -21138.801,E2 -21138.801} C_VEL
LIN {X 0,Y 222.176,Z 203.672,A -85,B 0,C 180,E1 -21139.336,E2 -21139.336} C_VEL
LIN {X 0,Y 219.548,Z 268.814,A -85,B 0,C 180,E1 -21141.428,E2 -21141.428} C_VEL
LIN {X 0,Y 218.628,Z 282.029,A -85,B 0,C 180,E1 -21142.206,E2 -21142.206} C_VEL
LIN {X 0,Y 217.363,Z 295.313,A -85,B 0,C 180,E1 -21143.386,E2 -21143.386} C_VEL
LIN {X 0,Y 215.711,Z 307.381,A -85,B 0,C 180,E1 -21144.86,E2 -21144.86} C_VEL
LIN {X 0,Y 213.826,Z 318.953,A -85,B 0,C 180,E1 -21146.703,E2 -21146.703} C_VEL
LIN {X 0,Y 211.981,Z 329.345,A -85,B 0,C 180,E1 -21148.813,E2 -21148.813} C_VEL
LIN {X 0,Y 209.871,Z 339.543,A -85,B 0,C 180,E1 -21151.439,E2 -21151.439} C_VEL
LIN {X 0,Y 208.09,Z 348.476,A -85,B 0,C 180,E1 -21154.359,E2 -21154.359} C_VEL
LIN {X 0,Y 206.686,Z 355.582,A -85,B 0,C 180,E1 -21157.326,E2 -21157.326} C_VEL
LIN {X 0,Y 205.471,Z 362.114,A -85,B 0,C 180,E1 -21160.844,E2 -21160.844} C_VEL
LIN {X 0,Y 204.807,Z 366.378,A -85,B 0,C 180,E1 -21163.899,E2 -21163.899} C_VEL
LIN {X 0,Y 204.466,Z 368.585,A -85,B 0,C 180,E1 -21165.961,E2 -21165.961} C_VEL
LIN {X 0,Y 204.303,Z 370.333,A -85,B 0,C 180,E1 -21168.035,E2 -21168.035} C_VEL
LIN {X 0,Y 204.38,Z 372.37,A -85,B 0,C 180,E1 -21171.807,E2 -21171.807} C_VEL
LIN {X 0,Y 204.68,Z 372.885,A -85,B 0,C 180,E1 -21174.333,E2 -21174.333} C_VEL
LIN {X 0,Y 205.339,Z 372.729,A -85,B 0,C 180,E1 -21177.142,E2 -21177.142} C_VEL
LIN {X 0,Y 206.653,Z 371.382,A -85,B 0,C 180,E1 -21180.673,E2 -21180.673} C_VEL
LIN {X 0,Y 207.73,Z 369.967,A -85,B 0,C 180,E1 -21182.774,E2 -21182.774} C_VEL
LIN {X 0,Y 209.627,Z 367.037,A -85,B 0,C 180,E1 -21185.762,E2 -21185.762} C_VEL
LIN {X 0,Y 212.218,Z 362.527,A -85,B 0,C 180,E1 -21188.993,E2 -21188.993} C_VEL
LIN {X 0,Y 215.204,Z 357.028,A -85,B 0,C 180,E1 -21191.901,E2 -21191.901} C_VEL
LIN {X 0,Y 218.96,Z 349.522,A -85,B 0,C 180,E1 -21194.922,E2 -21194.922} C_VEL
LIN {X 0,Y 222.307,Z 341.901,A -85,B 0,C 180,E1 -21197.31,E2 -21197.31} C_VEL
LIN {X 0,Y 226.123,Z 332.552,A -85,B 0,C 180,E1 -21199.58,E2 -21199.58} C_VEL
LIN {X 0,Y 229.834,Z 322.026,A -85,B 0,C 180,E1 -21201.59,E2 -21201.59} C_VEL
LIN {X 0,Y 232.954,Z 311.461,A -85,B 0,C 180,E1 -21203.17,E2 -21203.17} C_VEL
LIN {X 0,Y 235.694,Z 299.777,A -85,B 0,C 180,E1 -21204.53,E2 -21204.53} C_VEL
LIN {X 0,Y 237.991,Z 287.447,A -85,B 0,C 180,E1 -21205.59,E2 -21205.59} C_VEL
LIN {X 0,Y 239.609,Z 275.018,A -85,B 0,C 180,E1 -21206.346,E2 -21206.346} C_VEL
LIN {X 0,Y 240.78,Z 259.78,A -85,B 0,C 180,E1 -21206.884,E2 -21206.884} C_VEL
LIN {X 0,Y 242.844,Z 223.127,A -85,B 0,C 180,E1 -21207.955,E2 -21207.955} C_VEL
LIN {X 0,Y 236.82,Z 210.599,A -85,B 0,C 180,E1 -21210.005,E2 -21210.005} C_VEL
LIN {X 0,Y 230.088,Z 199.654,A -85,B 0,C 180,E1 -21212.419,E2 -21212.419} C_VEL
LIN {X 0,Y 224.032,Z 191.012,A -85,B 0,C 180,E1 -21214.77,E2 -21214.77} C_VEL
LIN {X 0,Y 221.334,Z 187.276,A -85,B 0,C 180,E1 -21215.897,E2 -21215.897} C_VEL
LIN {X 0,Y 218.084,Z 182.897,A -85,B 0,C 180,E1 -21217.351,E2 -21217.351} C_VEL
LIN {X 0,Y 215.422,Z 179.35,A -85,B 0,C 180,E1 -21218.62,E2 -21218.62} C_VEL
LIN {X 0,Y 214.621,Z 178.335,A -85,B 0,C 180,E1 -21219.013,E2 -21219.013} C_VEL
LIN {X 0,Y 212.196,Z 175.74,A -85,B 0,C 180,E1 -21220.218,E2 -21220.218} C_VEL
LIN {X 0,Y 210.764,Z 173.253,A -85,B 0,C 180,E1 -21221.028,E2 -21221.028} C_VEL
LIN {X 0,Y 208.409,Z 171.399,A -85,B 0,C 180,E1 -21222.269,E2 -21222.269} C_VEL
LIN {X 0,Y 207.005,Z 168.7,A -85,B 0,C 180,E1 -21223.164,E2 -21223.164} C_VEL
LIN {X 0,Y 206.818,Z 167.72,A -85,B 0,C 180,E1 -21223.402,E2 -21223.402} C_VEL
LIN {X 0,Y 206.902,Z 167.701,A -85,B 0,C 180,E1 -21228.241,E2 -21228.241} C_VEL
LIN {X 0,Y 207.129,Z 167.675,A -85,B 0,C 180,E1 -21232.2,E2 -21232.2} C_VEL
LIN {X 0,Y 207.342,Z 167.639,A -85,B 0,C 180,E1 -21238.058,E2 -21238.058} C_VEL
LIN {X 0,Y 207.481,Z 167.635,A -85,B 0,C 180,E1 -21240,E2 -21240} C_VEL
LIN {X 0,Y 207.345,Z 167.642,A -85,B 0,C 180,E1 -21241.943,E2 -21241.943} C_VEL
LIN {X 0,Y 207.127,Z 167.667,A -85,B 0,C 180,E1 -21247.801,E2 -21247.801} C_VEL
LIN {X 0,Y 206.919,Z 167.698,A -85,B 0,C 180,E1 -21251.759,E2 -21251.759} C_VEL
LIN {X 0,Y 206.846,Z 167.717,A -85,B 0,C 180,E1 -21255.773,E2 -21255.773} C_VEL
LIN {X 0,Y 206.859,Z 167.7,A -85,B 0,C 180,E1 -21257.955,E2 -21257.955} C_VEL
LIN {X 0,Y 206.748,Z 167.719,A -85,B 0,C 180,E1 -21263.391,E2 -21263.391} C_VEL
LIN {X 0,Y 206.719,Z 167.734,A -85,B 0,C 180,E1 -21268.423,E2 -21268.423} C_VEL
LIN {X 0,Y 206.767,Z 167.903,A -85,B 0,C 180,E1 -21271.61,E2 -21271.61} C_VEL
LIN {X 0,Y 208.31,Z 172.504,A -85,B 0,C 180,E1 -21275.931,E2 -21275.931} C_VEL
LIN {X 0,Y 209.072,Z 174.764,A -85,B 0,C 180,E1 -21277.7,E2 -21277.7} C_VEL
LIN {X 0,Y 212.212,Z 179.55,A -85,B 0,C 180,E1 -21279.454,E2 -21279.454} C_VEL
LIN {X 0,Y 213.995,Z 181.819,A -85,B 0,C 180,E1 -21280.362,E2 -21280.362} C_VEL
LIN {X 0,Y 217.629,Z 187.106,A -85,B 0,C 180,E1 -21282.142,E2 -21282.142} C_VEL
LIN {X 0,Y 221.264,Z 192.774,A -85,B 0,C 180,E1 -21283.796,E2 -21283.796} C_VEL
LIN {X 0,Y 223.955,Z 197.26,A -85,B 0,C 180,E1 -21284.95,E2 -21284.95} C_VEL
LIN {X 0,Y 225.064,Z 200.485,A -85,B 0,C 180,E1 -21285.482,E2 -21285.482} C_VEL
LIN {X 0,Y 226.755,Z 213.081,A -85,B 0,C 180,E1 -21286.66,E2 -21286.66} C_VEL
LIN {X 0,Y 227.983,Z 216.22,A -85,B 0,C 180,E1 -21287.189,E2 -21287.189} C_VEL
LIN {X 0,Y 233.268,Z 227.782,A -85,B 0,C 180,E1 -21289.253,E2 -21289.253} C_VEL
LIN {X 0,Y 235.54,Z 233.241,A -85,B 0,C 180,E1 -21290.103,E2 -21290.103} C_VEL
LIN {X 0,Y 236.713,Z 244.075,A -85,B 0,C 180,E1 -21290.881,E2 -21290.881} C_VEL
LIN {X 0,Y 234.087,Z 286.798,A -85,B 0,C 180,E1 -21292.196,E2 -21292.196} C_VEL
LIN {X 0,Y 232.338,Z 299.669,A -85,B 0,C 180,E1 -21292.84,E2 -21292.84} C_VEL
LIN {X 0,Y 229.97,Z 311.487,A -85,B 0,C 180,E1 -21293.693,E2 -21293.693} C_VEL
LIN {X 0,Y 227.109,Z 322.732,A -85,B 0,C 180,E1 -21294.805,E2 -21294.805} C_VEL
LIN {X 0,Y 223.473,Z 334.363,A -85,B 0,C 180,E1 -21296.338,E2 -21296.338} C_VEL
LIN {X 0,Y 220.167,Z 343.763,A -85,B 0,C 180,E1 -21297.947,E2 -21297.947} C_VEL
LIN {X 0,Y 216.613,Z 352.533,A -85,B 0,C 180,E1 -21299.808,E2 -21299.808} C_VEL
LIN {X 0,Y 212.95,Z 360.632,A -85,B 0,C 180,E1 -21301.946,E2 -21301.946} C_VEL
LIN {X 0,Y 208.993,Z 368.613,A -85,B 0,C 180,E1 -21304.611,E2 -21304.611} C_VEL
LIN {X 0,Y 206.001,Z 374.803,A -85,B 0,C 180,E1 -21307.299,E2 -21307.299} C_VEL
LIN {X 0,Y 203.502,Z 379.401,A -85,B 0,C 180,E1 -21309.796,E2 -21309.796} C_VEL
LIN {X 0,Y 201.168,Z 383.617,A -85,B 0,C 180,E1 -21312.725,E2 -21312.725} C_VEL
LIN {X 0,Y 199.332,Z 386.808,A -85,B 0,C 180,E1 -21315.711,E2 -21315.711} C_VEL
LIN {X 0,Y 197.941,Z 389.637,A -85,B 0,C 180,E1 -21319.774,E2 -21319.774} C_VEL
LIN {X 0,Y 197.336,Z 390.839,A -85,B 0,C 180,E1 -21323.866,E2 -21323.866} C_VEL
LIN {X 0,Y 197.356,Z 390.874,A -85,B 0,C 180,E1 -21325.915,E2 -21325.915} C_VEL
LIN {X 0,Y 197.478,Z 390.524,A -85,B 0,C 180,E1 -21327.96,E2 -21327.96} C_VEL
LIN {X 0,Y 197.612,Z 389.736,A -85,B 0,C 180,E1 -21330,E2 -21330} C_VEL
LIN {X 0,Y 197.496,Z 388.512,A -85,B 0,C 180,E1 -21332.039,E2 -21332.039} C_VEL
LIN {X 0,Y 197.408,Z 386.446,A -85,B 0,C 180,E1 -21334.552,E2 -21334.552} C_VEL
LIN {X 0,Y 197.582,Z 382.172,A -85,B 0,C 180,E1 -21338.179,E2 -21338.179} C_VEL
LIN {X 0,Y 198.105,Z 377.319,A -85,B 0,C 180,E1 -21341.251,E2 -21341.251} C_VEL
LIN {X 0,Y 199.071,Z 371.164,A -85,B 0,C 180,E1 -21344.307,E2 -21344.307} C_VEL
LIN {X 0,Y 200.54,Z 363.49,A -85,B 0,C 180,E1 -21347.33,E2 -21347.33} C_VEL
LIN {X 0,Y 202.061,Z 355.314,A -85,B 0,C 180,E1 -21349.907,E2 -21349.907} C_VEL
LIN {X 0,Y 204.381,Z 344.906,A -85,B 0,C 180,E1 -21352.492,E2 -21352.492} C_VEL
LIN {X 0,Y 206.462,Z 333.97,A -85,B 0,C 180,E1 -21354.644,E2 -21354.644} C_VEL
LIN {X 0,Y 208.34,Z 323.291,A -85,B 0,C 180,E1 -21356.279,E2 -21356.279} C_VEL
LIN {X 0,Y 210.103,Z 311.574,A -85,B 0,C 180,E1 -21357.653,E2 -21357.653} C_VEL
LIN {X 0,Y 211.649,Z 299.12,A -85,B 0,C 180,E1 -21358.714,E2 -21358.714} C_VEL
LIN {X 0,Y 212.637,Z 286.403,A -85,B 0,C 180,E1 -21359.448,E2 -21359.448} C_VEL
LIN {X 0,Y 214.513,Z 236.125,A -85,B 0,C 180,E1 -21361.138,E2 -21361.138} C_VEL
LIN {X 0,Y 210.699,Z 201.573,A -85,B 0,C 180,E1 -21362.929,E2 -21362.929} C_VEL
LIN {X 0,Y 203.801,Z 183.047,A -85,B 0,C 180,E1 -21364.609,E2 -21364.609} C_VEL
LIN {X 0,Y 201.803,Z 177.831,A -85,B 0,C 180,E1 -21365.167,E2 -21365.167} C_VEL
LIN {X 0,Y 199.676,Z 168.615,A -85,B 0,C 180,E1 -21369.557,E2 -21369.557} C_VEL
LIN {X 0,Y 199.581,Z 168.626,A -85,B 0,C 180,E1 -21375.228,E2 -21375.228} C_VEL
LIN {X 0,Y 199.58,Z 168.627,A -85,B 0,C 180,E1 -21378.005,E2 -21378.005} C_VEL
LIN {X 0,Y 199.611,Z 168.622,A -85,B 0,C 180,E1 -21380.767,E2 -21380.767} C_VEL
LIN {X 0,Y 199.615,Z 168.622,A -85,B 0,C 180,E1 -21385.713,E2 -21385.713} C_VEL
LIN {X 0,Y 199.702,Z 168.609,A -85,B 0,C 180,E1 -21388.137,E2 -21388.137} C_VEL
LIN {X 0,Y 199.687,Z 168.611,A -85,B 0,C 180,E1 -21392.771,E2 -21392.771} C_VEL
LIN {X 0,Y 199.713,Z 168.603,A -85,B 0,C 180,E1 -21397.226,E2 -21397.226} C_VEL
LIN {X 0,Y 199.748,Z 168.562,A -85,B 0,C 180,E1 -21401.8,E2 -21401.8} C_VEL
LIN {X 0,Y 199.813,Z 168.583,A -85,B 0,C 180,E1 -21405.746,E2 -21405.746} C_VEL
LIN {X 0,Y 200.022,Z 168.566,A -85,B 0,C 180,E1 -21409.881,E2 -21409.881} C_VEL
LIN {X 0,Y 200.011,Z 168.555,A -85,B 0,C 180,E1 -21413.949,E2 -21413.949} C_VEL
LIN {X 0,Y 200.319,Z 168.528,A -85,B 0,C 180,E1 -21417.989,E2 -21417.989} C_VEL
LIN {X 0,Y 200.479,Z 168.506,A -85,B 0,C 180,E1 -21420,E2 -21420} C_VEL
LIN {X 0,Y 200.027,Z 168.558,A -85,B 0,C 180,E1 -21424.029,E2 -21424.029} C_VEL
LIN {X 0,Y 200.089,Z 168.558,A -85,B 0,C 180,E1 -21428.076,E2 -21428.076} C_VEL
LIN {X 0,Y 199.874,Z 168.572,A -85,B 0,C 180,E1 -21432.179,E2 -21432.179} C_VEL
LIN {X 0,Y 199.804,Z 168.598,A -85,B 0,C 180,E1 -21436.343,E2 -21436.343} C_VEL
LIN {X 0,Y 199.69,Z 168.596,A -85,B 0,C 180,E1 -21440.606,E2 -21440.606} C_VEL
LIN {X 0,Y 199.664,Z 168.612,A -85,B 0,C 180,E1 -21444.985,E2 -21444.985} C_VEL
LIN {X 0,Y 199.663,Z 168.603,A -85,B 0,C 180,E1 -21449.524,E2 -21449.524} C_VEL
LIN {X 0,Y 199.67,Z 168.608,A -85,B 0,C 180,E1 -21452.355,E2 -21452.355} C_VEL
LIN {X 0,Y 199.622,Z 168.611,A -85,B 0,C 180,E1 -21456.763,E2 -21456.763} C_VEL
LIN {X 0,Y 199.607,Z 168.609,A -85,B 0,C 180,E1 -21459.328,E2 -21459.328} C_VEL
LIN {X 0,Y 199.573,Z 168.622,A -85,B 0,C 180,E1 -21462.31,E2 -21462.31} C_VEL
LIN {X 0,Y 199.578,Z 168.615,A -85,B 0,C 180,E1 -21465.229,E2 -21465.229} C_VEL
LIN {X 0,Y 199.579,Z 168.624,A -85,B 0,C 180,E1 -21468.005,E2 -21468.005} C_VEL
LIN {X 0,Y 199.609,Z 168.616,A -85,B 0,C 180,E1 -21470.768,E2 -21470.768} C_VEL
LIN {X 0,Y 199.613,Z 168.616,A -85,B 0,C 180,E1 -21475.714,E2 -21475.714} C_VEL
LIN {X 0,Y 199.7,Z 168.591,A -85,B 0,C 180,E1 -21478.137,E2 -21478.137} C_VEL
LIN {X 0,Y 199.686,Z 168.612,A -85,B 0,C 180,E1 -21482.772,E2 -21482.772} C_VEL
LIN {X 0,Y 199.712,Z 168.603,A -85,B 0,C 180,E1 -21487.226,E2 -21487.226} C_VEL
LIN {X 0,Y 199.794,Z 168.591,A -85,B 0,C 180,E1 -21491.759,E2 -21491.759} C_VEL
LIN {X 0,Y 199.809,Z 168.592,A -85,B 0,C 180,E1 -21494.94,E2 -21494.94} C_VEL
LIN {X 0,Y 200.837,Z 171.418,A -85,B 0,C 180,E1 -21495.218,E2 -21495.218} C_VEL
LIN {X 0,Y 210.066,Z 189.916,A -85,B 0,C 180,E1 -21497.288,E2 -21497.288} C_VEL
LIN {X 0,Y 213.888,Z 199.586,A -85,B 0,C 180,E1 -21498.157,E2 -21498.157} C_VEL
LIN {X 0,Y 215.66,Z 205.55,A -85,B 0,C 180,E1 -21498.606,E2 -21498.606} C_VEL
LIN {X 0,Y 212.97,Z 269.882,A -85,B 0,C 180,E1 -21500.743,E2 -21500.743} C_VEL
LIN {X 0,Y 211.986,Z 283.578,A -85,B 0,C 180,E1 -21501.6,E2 -21501.6} C_VEL
LIN {X 0,Y 210.654,Z 296.478,A -85,B 0,C 180,E1 -21502.813,E2 -21502.813} C_VEL
LIN {X 0,Y 209.047,Z 307.563,A -85,B 0,C 180,E1 -21504.212,E2 -21504.212} C_VEL
LIN {X 0,Y 207.081,Z 319.163,A -85,B 0,C 180,E1 -21506.108,E2 -21506.108} C_VEL
LIN {X 0,Y 205.346,Z 328.514,A -85,B 0,C 180,E1 -21508.039,E2 -21508.039} C_VEL
LIN {X 0,Y 203.388,Z 338.111,A -85,B 0,C 180,E1 -21510.495,E2 -21510.495} C_VEL
LIN {X 0,Y 201.655,Z 345.978,A -85,B 0,C 180,E1 -21512.997,E2 -21512.997} C_VEL
LIN {X 0,Y 200.096,Z 353.65,A -85,B 0,C 180,E1 -21516.049,E2 -21516.049} C_VEL
LIN {X 0,Y 198.831,Z 360.046,A -85,B 0,C 180,E1 -21519.277,E2 -21519.277} C_VEL
LIN {X 0,Y 198.018,Z 364.686,A -85,B 0,C 180,E1 -21522.296,E2 -21522.296} C_VEL
LIN {X 0,Y 197.38,Z 368.856,A -85,B 0,C 180,E1 -21525.978,E2 -21525.978} C_VEL
LIN {X 0,Y 197.192,Z 371.037,A -85,B 0,C 180,E1 -21528.709,E2 -21528.709} C_VEL
LIN {X 0,Y 197.329,Z 372.723,A -85,B 0,C 180,E1 -21532.18,E2 -21532.18} C_VEL
LIN {X 0,Y 197.746,Z 373.269,A -85,B 0,C 180,E1 -21535.245,E2 -21535.245} C_VEL
LIN {X 0,Y 198.412,Z 373.048,A -85,B 0,C 180,E1 -21537.684,E2 -21537.684} C_VEL
LIN {X 0,Y 200.082,Z 371.442,A -85,B 0,C 180,E1 -21541.796,E2 -21541.796} C_VEL
LIN {X 0,Y 201.933,Z 368.931,A -85,B 0,C 180,E1 -21545.048,E2 -21545.048} C_VEL
LIN {X 0,Y 204.35,Z 365.245,A -85,B 0,C 180,E1 -21548.248,E2 -21548.248} C_VEL
LIN {X 0,Y 207.08,Z 360.664,A -85,B 0,C 180,E1 -21551.161,E2 -21551.161} C_VEL
LIN {X 0,Y 210.872,Z 353.796,A -85,B 0,C 180,E1 -21554.419,E2 -21554.419} C_VEL
LIN {X 0,Y 214.221,Z 347.075,A -85,B 0,C 180,E1 -21556.884,E2 -21556.884} C_VEL
LIN {X 0,Y 217.939,Z 338.862,A -85,B 0,C 180,E1 -21559.273,E2 -21559.273} C_VEL
LIN {X 0,Y 221.649,Z 329.783,A -85,B 0,C 180,E1 -21561.335,E2 -21561.335} C_VEL
LIN {X 0,Y 225.128,Z 319.853,A -85,B 0,C 180,E1 -21563.126,E2 -21563.126} C_VEL
LIN {X 0,Y 228.589,Z 307.84,A -85,B 0,C 180,E1 -21564.829,E2 -21564.829} C_VEL
LIN {X 0,Y 231.277,Z 295.995,A -85,B 0,C 180,E1 -21566.096,E2 -21566.096} C_VEL
LIN {X 0,Y 233.573,Z 282.686,A -85,B 0,C 180,E1 -21567.112,E2 -21567.112} C_VEL
LIN {X 0,Y 235,Z 270.278,A -85,B 0,C 180,E1 -21567.748,E2 -21567.748} C_VEL
LIN {X 0,Y 237.71,Z 225.605,A -85,B 0,C 180,E1 -21569.099,E2 -21569.099} C_VEL
LIN {X 0,Y 232.254,Z 214.184,A -85,B 0,C 180,E1 -21571.086,E2 -21571.086} C_VEL
LIN {X 0,Y 225.975,Z 204.082,A -85,B 0,C 180,E1 -21573.456,E2 -21573.456} C_VEL
LIN {X 0,Y 220.652,Z 196.338,A -85,B 0,C 180,E1 -21575.633,E2 -21575.633} C_VEL
LIN {X 0,Y 217.831,Z 192.371,A -85,B 0,C 180,E1 -21576.889,E2 -21576.889} C_VEL
LIN {X 0,Y 215.132,Z 188.672,A -85,B 0,C 180,E1 -21578.162,E2 -21578.162} C_VEL
LIN {X 0,Y 211.962,Z 184.411,A -85,B 0,C 180,E1 -21579.753,E2 -21579.753} C_VEL
LIN {X 0,Y 209.393,Z 181.374,A -85,B 0,C 180,E1 -21581.105,E2 -21581.105} C_VEL
LIN {X 0,Y 208.49,Z 179.743,A -85,B 0,C 180,E1 -21581.641,E2 -21581.641} C_VEL
LIN {X 0,Y 205.874,Z 177.337,A -85,B 0,C 180,E1 -21583.102,E2 -21583.102} C_VEL
LIN {X 0,Y 204.136,Z 174.297,A -85,B 0,C 180,E1 -21584.269,E2 -21584.269} C_VEL
LIN {X 0,Y 201.605,Z 172.509,A -85,B 0,C 180,E1 -21585.876,E2 -21585.876} C_VEL
LIN {X 0,Y 200.138,Z 170.051,A -85,B 0,C 180,E1 -21587,E2 -21587} C_VEL
LIN {X 0,Y 199.831,Z 168.59,A -85,B 0,C 180,E1 -21587.432,E2 -21587.432} C_VEL
LIN {X 0,Y 200.025,Z 168.556,A -85,B 0,C 180,E1 -21589.882,E2 -21589.882} C_VEL
LIN {X 0,Y 200.001,Z 168.555,A -85,B 0,C 180,E1 -21593.949,E2 -21593.949} C_VEL
LIN {X 0,Y 200.284,Z 168.518,A -85,B 0,C 180,E1 -21597.989,E2 -21597.989} C_VEL
LIN {X 0,Y 200.448,Z 168.51,A -85,B 0,C 180,E1 -21600,E2 -21600} C_VEL
LIN {X 0,Y 199.99,Z 168.558,A -85,B 0,C 180,E1 -21604.031,E2 -21604.031} C_VEL
LIN {X 0,Y 200.075,Z 168.545,A -85,B 0,C 180,E1 -21608.078,E2 -21608.078} C_VEL
LIN {X 0,Y 199.869,Z 168.573,A -85,B 0,C 180,E1 -21612.18,E2 -21612.18} C_VEL
LIN {X 0,Y 199.79,Z 168.588,A -85,B 0,C 180,E1 -21616.345,E2 -21616.345} C_VEL
LIN {X 0,Y 199.677,Z 168.606,A -85,B 0,C 180,E1 -21620.608,E2 -21620.608} C_VEL
LIN {X 0,Y 199.653,Z 168.61,A -85,B 0,C 180,E1 -21624.988,E2 -21624.988} C_VEL
LIN {X 0,Y 199.693,Z 168.679,A -85,B 0,C 180,E1 -21627.996,E2 -21627.996} C_VEL
LIN {X 0,Y 200.817,Z 171.91,A -85,B 0,C 180,E1 -21631.666,E2 -21631.666} C_VEL
LIN {X 0,Y 201.581,Z 174.05,A -85,B 0,C 180,E1 -21633.658,E2 -21633.658} C_VEL
LIN {X 0,Y 205.356,Z 179.489,A -85,B 0,C 180,E1 -21636.205,E2 -21636.205} C_VEL
LIN {X 0,Y 206.783,Z 181.273,A -85,B 0,C 180,E1 -21637.054,E2 -21637.054} C_VEL
LIN {X 0,Y 210.518,Z 186.616,A -85,B 0,C 180,E1 -21639.173,E2 -21639.173} C_VEL
LIN {X 0,Y 215.518,Z 194.333,A -85,B 0,C 180,E1 -21641.754,E2 -21641.754} C_VEL
LIN {X 0,Y 219.254,Z 200.403,A -85,B 0,C 180,E1 -21643.514,E2 -21643.514} C_VEL
LIN {X 0,Y 224.282,Z 209.129,A -85,B 0,C 180,E1 -21645.682,E2 -21645.682} C_VEL
LIN {X 0,Y 227.983,Z 216.22,A -85,B 0,C 180,E1 -21647.189,E2 -21647.189} C_VEL
LIN {X 0,Y 229.426,Z 219.153,A -85,B 0,C 180,E1 -21647.76,E2 -21647.76} C_VEL
LIN {X 0,Y 230.905,Z 224.296,A -85,B 0,C 180,E1 -21648.433,E2 -21648.433} C_VEL
LIN {X 0,Y 231.832,Z 231.942,A -85,B 0,C 180,E1 -21649.055,E2 -21649.055} C_VEL
LIN {X 0,Y 231.962,Z 238.027,A -85,B 0,C 180,E1 -21649.377,E2 -21649.377} C_VEL
LIN {X 0,Y 231.693,Z 246.242,A -85,B 0,C 180,E1 -21649.688,E2 -21649.688} C_VEL
LIN {X 0,Y 229.121,Z 286.111,A -85,B 0,C 180,E1 -21650.93,E2 -21650.93} C_VEL
LIN {X 0,Y 227.325,Z 299.029,A -85,B 0,C 180,E1 -21651.574,E2 -21651.574} C_VEL
LIN {X 0,Y 224.826,Z 311.088,A -85,B 0,C 180,E1 -21652.442,E2 -21652.442} C_VEL
LIN {X 0,Y 221.89,Z 322.344,A -85,B 0,C 180,E1 -21653.567,E2 -21653.567} C_VEL
LIN {X 0,Y 218.076,Z 333.994,A -85,B 0,C 180,E1 -21655.107,E2 -21655.107} C_VEL
LIN {X 0,Y 214.208,Z 344.464,A -85,B 0,C 180,E1 -21656.944,E2 -21656.944} C_VEL
LIN {X 0,Y 210.538,Z 353.063,A -85,B 0,C 180,E1 -21658.841,E2 -21658.841} C_VEL
LIN {X 0,Y 206.716,Z 361.021,A -85,B 0,C 180,E1 -21661.021,E2 -21661.021} C_VEL
LIN {X 0,Y 202.619,Z 368.863,A -85,B 0,C 180,E1 -21663.752,E2 -21663.752} C_VEL
LIN {X 0,Y 199.65,Z 374.427,A -85,B 0,C 180,E1 -21666.241,E2 -21666.241} C_VEL
LIN {X 0,Y 196.844,Z 379.464,A -85,B 0,C 180,E1 -21669.081,E2 -21669.081} C_VEL
LIN {X 0,Y 194.386,Z 383.591,A -85,B 0,C 180,E1 -21672.102,E2 -21672.102} C_VEL
LIN {X 0,Y 192.425,Z 386.697,A -85,B 0,C 180,E1 -21675.187,E2 -21675.187} C_VEL
LIN {X 0,Y 191.582,Z 388.27,A -85,B 0,C 180,E1 -21677.284,E2 -21677.284} C_VEL
LIN {X 0,Y 190.484,Z 390.157,A -85,B 0,C 180,E1 -21681.513,E2 -21681.513} C_VEL
LIN {X 0,Y 190.278,Z 390.53,A -85,B 0,C 180,E1 -21685.763,E2 -21685.763} C_VEL
LIN {X 0,Y 190.391,Z 390.121,A -85,B 0,C 180,E1 -21687.884,E2 -21687.884} C_VEL
LIN {X 0,Y 190.546,Z 389.286,A -85,B 0,C 180,E1 -21690,E2 -21690} C_VEL
LIN {X 0,Y 190.411,Z 388.026,A -85,B 0,C 180,E1 -21692.115,E2 -21692.115} C_VEL
LIN {X 0,Y 190.337,Z 386.134,A -85,B 0,C 180,E1 -21694.473,E2 -21694.473} C_VEL
LIN {X 0,Y 190.427,Z 382.926,A -85,B 0,C 180,E1 -21697.421,E2 -21697.421} C_VEL
LIN {X 0,Y 190.862,Z 378.39,A -85,B 0,C 180,E1 -21700.609,E2 -21700.609} C_VEL
LIN {X 0,Y 191.943,Z 371.47,A -85,B 0,C 180,E1 -21704.309,E2 -21704.309} C_VEL
LIN {X 0,Y 193.429,Z 363.928,A -85,B 0,C 180,E1 -21707.442,E2 -21707.442} C_VEL
LIN {X 0,Y 194.795,Z 356.893,A -85,B 0,C 180,E1 -21709.813,E2 -21709.813} C_VEL
LIN {X 0,Y 197.139,Z 346.859,A -85,B 0,C 180,E1 -21712.534,E2 -21712.534} C_VEL
LIN {X 0,Y 198.981,Z 337.698,A -85,B 0,C 180,E1 -21714.519,E2 -21714.519} C_VEL
LIN {X 0,Y 200.832,Z 327.978,A -85,B 0,C 180,E1 -21716.219,E2 -21716.219} C_VEL
LIN {X 0,Y 202.891,Z 315.686,A -85,B 0,C 180,E1 -21717.88,E2 -21717.88} C_VEL
LIN {X 0,Y 204.685,Z 302.834,A -85,B 0,C 180,E1 -21719.152,E2 -21719.152} C_VEL
LIN {X 0,Y 205.852,Z 289.877,A -85,B 0,C 180,E1 -21720.025,E2 -21720.025} C_VEL
LIN {X 0,Y 206.752,Z 272.38,A -85,B 0,C 180,E1 -21720.704,E2 -21720.704} C_VEL
LIN {X 0,Y 208.045,Z 236.582,A -85,B 0,C 180,E1 -21721.923,E2 -21721.923} C_VEL
LIN {X 0,Y 204.455,Z 203.547,A -85,B 0,C 180,E1 -21723.695,E2 -21723.695} C_VEL
LIN {X 0,Y 197.231,Z 184.282,A -85,B 0,C 180,E1 -21725.55,E2 -21725.55} C_VEL
LIN {X 0,Y 194.505,Z 177.589,A -85,B 0,C 180,E1 -21726.276,E2 -21726.276} C_VEL
LIN {X 0,Y 192.598,Z 169.494,A -85,B 0,C 180,E1 -21730.274,E2 -21730.274} C_VEL
LIN {X 0,Y 192.493,Z 169.51,A -85,B 0,C 180,E1 -21736.076,E2 -21736.076} C_VEL
LIN {X 0,Y 192.519,Z 169.507,A -85,B 0,C 180,E1 -21740.05,E2 -21740.05} C_VEL
LIN {X 0,Y 192.561,Z 169.5,A -85,B 0,C 180,E1 -21744.27,E2 -21744.27} C_VEL
LIN {X 0,Y 192.612,Z 169.494,A -85,B 0,C 180,E1 -21747.057,E2 -21747.057} C_VEL
LIN {X 0,Y 192.665,Z 169.486,A -85,B 0,C 180,E1 -21751.691,E2 -21751.691} C_VEL
LIN {X 0,Y 192.685,Z 169.481,A -85,B 0,C 180,E1 -21756.345,E2 -21756.345} C_VEL
LIN {X 0,Y 192.697,Z 169.44,A -85,B 0,C 180,E1 -21761.489,E2 -21761.489} C_VEL
LIN {X 0,Y 192.739,Z 169.457,A -85,B 0,C 180,E1 -21765.211,E2 -21765.211} C_VEL
LIN {X 0,Y 192.945,Z 169.448,A -85,B 0,C 180,E1 -21769.566,E2 -21769.566} C_VEL
LIN {X 0,Y 192.974,Z 169.431,A -85,B 0,C 180,E1 -21773.727,E2 -21773.727} C_VEL
LIN {X 0,Y 193.26,Z 169.407,A -85,B 0,C 180,E1 -21777.916,E2 -21777.916} C_VEL
LIN {X 0,Y 193.443,Z 169.382,A -85,B 0,C 180,E1 -21780,E2 -21780} C_VEL
LIN {X 0,Y 192.973,Z 169.437,A -85,B 0,C 180,E1 -21784.177,E2 -21784.177} C_VEL
LIN {X 0,Y 193.036,Z 169.435,A -85,B 0,C 180,E1 -21788.373,E2 -21788.373} C_VEL
LIN {X 0,Y 192.802,Z 169.455,A -85,B 0,C 180,E1 -21792.633,E2 -21792.633} C_VEL
LIN {X 0,Y 192.757,Z 169.472,A -85,B 0,C 180,E1 -21796.958,E2 -21796.958} C_VEL
LIN {X 0,Y 192.621,Z 169.475,A -85,B 0,C 180,E1 -21801.399,E2 -21801.399} C_VEL
LIN {X 0,Y 192.646,Z 169.486,A -85,B 0,C 180,E1 -21804.213,E2 -21804.213} C_VEL
LIN {X 0,Y 192.643,Z 169.479,A -85,B 0,C 180,E1 -21808.889,E2 -21808.889} C_VEL
LIN {X 0,Y 192.596,Z 169.489,A -85,B 0,C 180,E1 -21813.186,E2 -21813.186} C_VEL
LIN {X 0,Y 192.55,Z 169.486,A -85,B 0,C 180,E1 -21818.352,E2 -21818.352} C_VEL
LIN {X 0,Y 192.49,Z 169.504,A -85,B 0,C 180,E1 -21823.096,E2 -21823.096} C_VEL
LIN {X 0,Y 192.49,Z 169.502,A -85,B 0,C 180,E1 -21826.904,E2 -21826.904} C_VEL
LIN {X 0,Y 192.55,Z 169.494,A -85,B 0,C 180,E1 -21831.648,E2 -21831.648} C_VEL
LIN {X 0,Y 192.598,Z 169.484,A -85,B 0,C 180,E1 -21836.815,E2 -21836.815} C_VEL
LIN {X 0,Y 192.664,Z 169.487,A -85,B 0,C 180,E1 -21841.692,E2 -21841.692} C_VEL
LIN {X 0,Y 192.684,Z 169.472,A -85,B 0,C 180,E1 -21846.346,E2 -21846.346} C_VEL
LIN {X 0,Y 192.729,Z 169.47,A -85,B 0,C 180,E1 -21851.46,E2 -21851.46} C_VEL
LIN {X 0,Y 192.776,Z 169.63,A -85,B 0,C 180,E1 -21853.843,E2 -21853.843} C_VEL
LIN {X 0,Y 193.89,Z 172.501,A -85,B 0,C 180,E1 -21854.153,E2 -21854.153} C_VEL
LIN {X 0,Y 201.953,Z 188.351,A -85,B 0,C 180,E1 -21856.084,E2 -21856.084} C_VEL
LIN {X 0,Y 206.947,Z 199.682,A -85,B 0,C 180,E1 -21857.246,E2 -21857.246} C_VEL
LIN {X 0,Y 209.194,Z 207.007,A -85,B 0,C 180,E1 -21857.833,E2 -21857.833} C_VEL
LIN {X 0,Y 206.45,Z 270.235,A -85,B 0,C 180,E1 -21859.991,E2 -21859.991} C_VEL
LIN {X 0,Y 205.438,Z 283.478,A -85,B 0,C 180,E1 -21860.835,E2 -21860.835} C_VEL
LIN {X 0,Y 204.086,Z 296.505,A -85,B 0,C 180,E1 -21862.083,E2 -21862.083} C_VEL
LIN {X 0,Y 202.421,Z 307.65,A -85,B 0,C 180,E1 -21863.521,E2 -21863.521} C_VEL
LIN {X 0,Y 200.352,Z 319.305,A -85,B 0,C 180,E1 -21865.474,E2 -21865.474} C_VEL
LIN {X 0,Y 198.339,Z 329.768,A -85,B 0,C 180,E1 -21867.716,E2 -21867.716} C_VEL
LIN {X 0,Y 196.521,Z 338.319,A -85,B 0,C 180,E1 -21870,E2 -21870} C_VEL
LIN {X 0,Y 194.703,Z 346.21,A -85,B 0,C 180,E1 -21872.586,E2 -21872.586} C_VEL
LIN {X 0,Y 193.106,Z 353.895,A -85,B 0,C 180,E1 -21875.744,E2 -21875.744} C_VEL
LIN {X 0,Y 191.675,Z 360.82,A -85,B 0,C 180,E1 -21879.391,E2 -21879.391} C_VEL
LIN {X 0,Y 190.809,Z 365.652,A -85,B 0,C 180,E1 -21882.768,E2 -21882.768} C_VEL
LIN {X 0,Y 190.272,Z 369.279,A -85,B 0,C 180,E1 -21886.189,E2 -21886.189} C_VEL
LIN {X 0,Y 190.072,Z 371.666,A -85,B 0,C 180,E1 -21889.438,E2 -21889.438} C_VEL
LIN {X 0,Y 190.274,Z 373.067,A -85,B 0,C 180,E1 -21892.572,E2 -21892.572} C_VEL
LIN {X 0,Y 190.874,Z 373.591,A -85,B 0,C 180,E1 -21896.222,E2 -21896.222} C_VEL
LIN {X 0,Y 191.571,Z 373.326,A -85,B 0,C 180,E1 -21898.485,E2 -21898.485} C_VEL
LIN {X 0,Y 192.443,Z 372.635,A -85,B 0,C 180,E1 -21900.75,E2 -21900.75} C_VEL
LIN {X 0,Y 193.845,Z 371.104,A -85,B 0,C 180,E1 -21903.501,E2 -21903.501} C_VEL
LIN {X 0,Y 196.47,Z 367.619,A -85,B 0,C 180,E1 -21907.454,E2 -21907.454} C_VEL
LIN {X 0,Y 199.304,Z 363.309,A -85,B 0,C 180,E1 -21910.72,E2 -21910.72} C_VEL
LIN {X 0,Y 202.779,Z 357.626,A -85,B 0,C 180,E1 -21913.882,E2 -21913.882} C_VEL
LIN {X 0,Y 206.381,Z 351.197,A -85,B 0,C 180,E1 -21916.622,E2 -21916.622} C_VEL
LIN {X 0,Y 210.529,Z 342.811,A -85,B 0,C 180,E1 -21919.416,E2 -21919.416} C_VEL
LIN {X 0,Y 214.725,Z 333.484,A -85,B 0,C 180,E1 -21921.77,E2 -21921.77} C_VEL
LIN {X 0,Y 218.691,Z 323.131,A -85,B 0,C 180,E1 -21923.825,E2 -21923.825} C_VEL
LIN {X 0,Y 221.994,Z 313.01,A -85,B 0,C 180,E1 -21925.399,E2 -21925.399} C_VEL
LIN {X 0,Y 225.081,Z 301.104,A -85,B 0,C 180,E1 -21926.846,E2 -21926.846} C_VEL
LIN {X 0,Y 227.718,Z 288.196,A -85,B 0,C 180,E1 -21927.989,E2 -21927.989} C_VEL
LIN {X 0,Y 229.469,Z 276.015,A -85,B 0,C 180,E1 -21928.747,E2 -21928.747} C_VEL
LIN {X 0,Y 230.694,Z 261.734,A -85,B 0,C 180,E1 -21929.276,E2 -21929.276} C_VEL
LIN {X 0,Y 232.83,Z 228.428,A -85,B 0,C 180,E1 -21930.253,E2 -21930.253} C_VEL
LIN {X 0,Y 228.322,Z 218.942,A -85,B 0,C 180,E1 -21931.99,E2 -21931.99} C_VEL
LIN {X 0,Y 222.632,Z 209.514,A -85,B 0,C 180,E1 -21934.248,E2 -21934.248} C_VEL
LIN {X 0,Y 217.246,Z 201.486,A -85,B 0,C 180,E1 -21936.576,E2 -21936.576} C_VEL
LIN {X 0,Y 212.353,Z 194.519,A -85,B 0,C 180,E1 -21938.937,E2 -21938.937} C_VEL
LIN {X 0,Y 209.235,Z 190.383,A -85,B 0,C 180,E1 -21940.565,E2 -21940.565} C_VEL
LIN {X 0,Y 206.501,Z 186.797,A -85,B 0,C 180,E1 -21942.1,E2 -21942.1} C_VEL
LIN {X 0,Y 205.443,Z 185.561,A -85,B 0,C 180,E1 -21942.714,E2 -21942.714} C_VEL
LIN {X 0,Y 202.999,Z 182.582,A -85,B 0,C 180,E1 -21944.243,E2 -21944.243} C_VEL
LIN {X 0,Y 201.92,Z 180.821,A -85,B 0,C 180,E1 -21944.997,E2 -21944.997} C_VEL
LIN {X 0,Y 199.337,Z 178.56,A -85,B 0,C 180,E1 -21946.752,E2 -21946.752} C_VEL
LIN {X 0,Y 197.732,Z 175.592,A -85,B 0,C 180,E1 -21948.078,E2 -21948.078} C_VEL
LIN {X 0,Y 194.564,Z 173.082,A -85,B 0,C 180,E1 -21950.646,E2 -21950.646} C_VEL
LIN {X 0,Y 193.355,Z 170.842,A -85,B 0,C 180,E1 -21951.904,E2 -21951.904} C_VEL
LIN {X 0,Y 193.004,Z 169.431,A -85,B 0,C 180,E1 -21952.415,E2 -21952.415} C_VEL
LIN {X 0,Y 193.229,Z 169.397,A -85,B 0,C 180,E1 -21957.916,E2 -21957.916} C_VEL
LIN {X 0,Y 193.415,Z 169.385,A -85,B 0,C 180,E1 -21960,E2 -21960} C_VEL
LIN {X 0,Y 192.937,Z 169.438,A -85,B 0,C 180,E1 -21964.178,E2 -21964.178} C_VEL
LIN {X 0,Y 193.026,Z 169.423,A -85,B 0,C 180,E1 -21968.375,E2 -21968.375} C_VEL
LIN {X 0,Y 192.796,Z 169.452,A -85,B 0,C 180,E1 -21972.634,E2 -21972.634} C_VEL
LIN {X 0,Y 192.749,Z 169.46,A -85,B 0,C 180,E1 -21976.96,E2 -21976.96} C_VEL
LIN {X 0,Y 192.659,Z 169.469,A -85,B 0,C 180,E1 -21982.522,E2 -21982.522} C_VEL
LIN {X 0,Y 192.702,Z 169.662,A -85,B 0,C 180,E1 -21983.652,E2 -21983.652} C_VEL
LIN {X 0,Y 193.907,Z 172.985,A -85,B 0,C 180,E1 -21988.228,E2 -21988.228} C_VEL
LIN {X 0,Y 195.935,Z 176.358,A -85,B 0,C 180,E1 -21990.144,E2 -21990.144} C_VEL
LIN {X 0,Y 199.694,Z 180.742,A -85,B 0,C 180,E1 -21993.08,E2 -21993.08} C_VEL
LIN {X 0,Y 203.578,Z 186.261,A -85,B 0,C 180,E1 -21995.784,E2 -21995.784} C_VEL
LIN {X 0,Y 208.744,Z 193.957,A -85,B 0,C 180,E1 -21998.867,E2 -21998.867} C_VEL
LIN {X 0,Y 212.645,Z 200.126,A -85,B 0,C 180,E1 -22000.954,E2 -22000.954} C_VEL
LIN {X 0,Y 216.461,Z 206.566,A -85,B 0,C 180,E1 -22002.845,E2 -22002.845} C_VEL
LIN {X 0,Y 222.349,Z 217.268,A -85,B 0,C 180,E1 -22005.485,E2 -22005.485} C_VEL
LIN {X 0,Y 228.027,Z 229.405,A -85,B 0,C 180,E1 -22007.854,E2 -22007.854} C_VEL
LIN {X 0,Y 230.969,Z 237.047,A -85,B 0,C 180,E1 -22009.058,E2 -22009.058} C_VEL
LIN {X 0,Y 231.772,Z 244.782,A -85,B 0,C 180,E1 -22009.641,E2 -22009.641} C_VEL
LIN {X 0,Y 231.693,Z 246.242,A -85,B 0,C 180,E1 -22009.688,E2 -22009.688} C_VEL
LIN {X 0,Y 230.937,Z 252.088,A -85,B 0,C 180,E1 -22009.757,E2 -22009.757} C_VEL
LIN {X 0,Y 225.864,Z 271.181,A -85,B 0,C 180,E1 -22009.268,E2 -22009.268} C_VEL
LIN {X 0,Y 225.009,Z 277.037,A -85,B 0,C 180,E1 -22009.312,E2 -22009.312} C_VEL
LIN {X 0,Y 223.637,Z 291.051,A -85,B 0,C 180,E1 -22009.838,E2 -22009.838} C_VEL
LIN {X 0,Y 221.431,Z 303.799,A -85,B 0,C 180,E1 -22010.596,E2 -22010.596} C_VEL
LIN {X 0,Y 218.788,Z 314.857,A -85,B 0,C 180,E1 -22011.51,E2 -22011.51} C_VEL
LIN {X 0,Y 215.253,Z 326.758,A -85,B 0,C 180,E1 -22012.841,E2 -22012.841} C_VEL
LIN {X 0,Y 211.412,Z 337.428,A -85,B 0,C 180,E1 -22014.426,E2 -22014.426} C_VEL
LIN {X 0,Y 207.888,Z 346.187,A -85,B 0,C 180,E1 -22016.095,E2 -22016.095} C_VEL
LIN {X 0,Y 203.725,Z 355.246,A -85,B 0,C 180,E1 -22018.258,E2 -22018.258} C_VEL
LIN {X 0,Y 199.055,Z 364.133,A -85,B 0,C 180,E1 -22020.956,E2 -22020.956} C_VEL
LIN {X 0,Y 194.991,Z 371.314,A -85,B 0,C 180,E1 -22023.798,E2 -22023.798} C_VEL
LIN {X 0,Y 191.239,Z 377.9,A -85,B 0,C 180,E1 -22027.302,E2 -22027.302} C_VEL
LIN {X 0,Y 188.428,Z 382.304,A -85,B 0,C 180,E1 -22030.386,E2 -22030.386} C_VEL
LIN {X 0,Y 185.537,Z 386.587,A -85,B 0,C 180,E1 -22034.623,E2 -22034.623} C_VEL
LIN {X 0,Y 184.626,Z 388.088,A -85,B 0,C 180,E1 -22036.797,E2 -22036.797} C_VEL
LIN {X 0,Y 183.435,Z 389.888,A -85,B 0,C 180,E1 -22041.184,E2 -22041.184} C_VEL
LIN {X 0,Y 183.187,Z 390.174,A -85,B 0,C 180,E1 -22045.599,E2 -22045.599} C_VEL
LIN {X 0,Y 183.307,Z 389.698,A -85,B 0,C 180,E1 -22047.802,E2 -22047.802} C_VEL
LIN {X 0,Y 183.481,Z 388.826,A -85,B 0,C 180,E1 -22050,E2 -22050} C_VEL
LIN {X 0,Y 183.328,Z 387.524,A -85,B 0,C 180,E1 -22052.197,E2 -22052.197} C_VEL
LIN {X 0,Y 183.247,Z 384.721,A -85,B 0,C 180,E1 -22055.502,E2 -22055.502} C_VEL
LIN {X 0,Y 183.492,Z 380.854,A -85,B 0,C 180,E1 -22058.812,E2 -22058.812} C_VEL
LIN {X 0,Y 184.125,Z 375.817,A -85,B 0,C 180,E1 -22062.118,E2 -22062.118} C_VEL
LIN {X 0,Y 185.28,Z 369.461,A -85,B 0,C 180,E1 -22065.398,E2 -22065.398} C_VEL
LIN {X 0,Y 186.945,Z 361.462,A -85,B 0,C 180,E1 -22068.635,E2 -22068.635} C_VEL
LIN {X 0,Y 188.789,Z 352.708,A -85,B 0,C 180,E1 -22071.46,E2 -22071.46} C_VEL
LIN {X 0,Y 190.936,Z 343.294,A -85,B 0,C 180,E1 -22073.884,E2 -22073.884} C_VEL
LIN {X 0,Y 192.967,Z 333.47,A -85,B 0,C 180,E1 -22075.915,E2 -22075.915} C_VEL
LIN {X 0,Y 195.009,Z 322.842,A -85,B 0,C 180,E1 -22077.645,E2 -22077.645} C_VEL
LIN {X 0,Y 197.076,Z 310.046,A -85,B 0,C 180,E1 -22079.216,E2 -22079.216} C_VEL
LIN {X 0,Y 198.688,Z 297.257,A -85,B 0,C 180,E1 -22080.341,E2 -22080.341} C_VEL
LIN {X 0,Y 199.716,Z 284.942,A -85,B 0,C 180,E1 -22081.047,E2 -22081.047} C_VEL
LIN {X 0,Y 201.591,Z 237.117,A -85,B 0,C 180,E1 -22082.747,E2 -22082.747} C_VEL
LIN {X 0,Y 198.286,Z 205.741,A -85,B 0,C 180,E1 -22084.494,E2 -22084.494} C_VEL
LIN {X 0,Y 191.381,Z 187.209,A -85,B 0,C 180,E1 -22086.369,E2 -22086.369} C_VEL
LIN {X 0,Y 187.168,Z 177.186,A -85,B 0,C 180,E1 -22087.567,E2 -22087.567} C_VEL
LIN {X 0,Y 185.529,Z 170.375,A -85,B 0,C 180,E1 -22091.133,E2 -22091.133} C_VEL
LIN {X 0,Y 185.461,Z 170.386,A -85,B 0,C 180,E1 -22096.054,E2 -22096.054} C_VEL
LIN {X 0,Y 185.469,Z 170.386,A -85,B 0,C 180,E1 -22099.895,E2 -22099.895} C_VEL
LIN {X 0,Y 185.507,Z 170.379,A -85,B 0,C 180,E1 -22102.711,E2 -22102.711} C_VEL
LIN {X 0,Y 185.547,Z 170.373,A -85,B 0,C 180,E1 -22107.975,E2 -22107.975} C_VEL
LIN {X 0,Y 185.583,Z 170.368,A -85,B 0,C 180,E1 -22110.575,E2 -22110.575} C_VEL
LIN {X 0,Y 185.58,Z 170.369,A -85,B 0,C 180,E1 -22115.381,E2 -22115.381} C_VEL
LIN {X 0,Y 185.584,Z 170.337,A -85,B 0,C 180,E1 -22120.072,E2 -22120.072} C_VEL
LIN {X 0,Y 185.668,Z 170.333,A -85,B 0,C 180,E1 -22124.634,E2 -22124.634} C_VEL
LIN {X 0,Y 185.888,Z 170.328,A -85,B 0,C 180,E1 -22129.418,E2 -22129.418} C_VEL
LIN {X 0,Y 185.937,Z 170.307,A -85,B 0,C 180,E1 -22133.489,E2 -22133.489} C_VEL
LIN {X 0,Y 186.204,Z 170.286,A -85,B 0,C 180,E1 -22137.836,E2 -22137.836} C_VEL
LIN {X 0,Y 186.406,Z 170.259,A -85,B 0,C 180,E1 -22140,E2 -22140} C_VEL
LIN {X 0,Y 185.92,Z 170.315,A -85,B 0,C 180,E1 -22144.335,E2 -22144.335} C_VEL
LIN {X 0,Y 185.983,Z 170.311,A -85,B 0,C 180,E1 -22148.693,E2 -22148.693} C_VEL
LIN {X 0,Y 185.729,Z 170.34,A -85,B 0,C 180,E1 -22153.122,E2 -22153.122} C_VEL
LIN {X 0,Y 185.69,Z 170.353,A -85,B 0,C 180,E1 -22157.625,E2 -22157.625} C_VEL
LIN {X 0,Y 185.58,Z 170.355,A -85,B 0,C 180,E1 -22162.253,E2 -22162.253} C_VEL
LIN {X 0,Y 185.558,Z 170.368,A -85,B 0,C 180,E1 -22167.032,E2 -22167.032} C_VEL
LIN {X 0,Y 185.576,Z 170.356,A -85,B 0,C 180,E1 -22169.493,E2 -22169.493} C_VEL
LIN {X 0,Y 185.498,Z 170.375,A -85,B 0,C 180,E1 -22174.632,E2 -22174.632} C_VEL
LIN {X 0,Y 185.505,Z 170.367,A -85,B 0,C 180,E1 -22177.313,E2 -22177.313} C_VEL
LIN {X 0,Y 185.47,Z 170.377,A -85,B 0,C 180,E1 -22180.725,E2 -22180.725} C_VEL
LIN {X 0,Y 185.459,Z 170.374,A -85,B 0,C 180,E1 -22186.055,E2 -22186.055} C_VEL
LIN {X 0,Y 185.467,Z 170.379,A -85,B 0,C 180,E1 -22189.896,E2 -22189.896} C_VEL
LIN {X 0,Y 185.505,Z 170.374,A -85,B 0,C 180,E1 -22192.711,E2 -22192.711} C_VEL
LIN {X 0,Y 185.545,Z 170.353,A -85,B 0,C 180,E1 -22197.976,E2 -22197.976} C_VEL
LIN {X 0,Y 185.581,Z 170.362,A -85,B 0,C 180,E1 -22200.576,E2 -22200.576} C_VEL
LIN {X 0,Y 185.579,Z 170.356,A -85,B 0,C 180,E1 -22205.382,E2 -22205.382} C_VEL
LIN {X 0,Y 185.672,Z 170.349,A -85,B 0,C 180,E1 -22211.136,E2 -22211.136} C_VEL
